LIN {X -0.262,Y -467.688,Z 682.023,A 0.000,B 0.000,C 90.000,E1 220.092} C_DIS
LIN {X -0.082,Y -463.648,Z 682.012,A 0.000,B 0.000,C 90.000,E1 218.177} C_DIS
LIN {X -0.203,Y -456.849,Z 681.993,A 0.000,B 0.000,C 90.000,E1 214.692} C_DIS
LIN {X -0.182,Y -453.797,Z 681.984,A 0.000,B 0.000,C 90.000,E1 213.086} C_DIS
LIN {X -0.004,Y -450.100,Z 681.973,A 0.000,B 0.000,C 90.000,E1 211.131} C_DIS
LIN {X -0.145,Y -446.430,Z 681.962,A 0.000,B 0.000,C 90.000,E1 209.205} C_DIS
LIN {X -0.102,Y -444.091,Z 681.955,A 0.000,B 0.000,C 90.000,E1 207.897} C_DIS
LIN {X 0.139,Y -441.158,Z 681.946,A 0.000,B 0.000,C 90.000,E1 206.232} C_DIS
LIN {X -0.011,Y -437.014,Z 681.933,A 0.000,B 0.000,C 90.000,E1 203.951} C_DIS
LIN {X -0.104,Y -434.577,Z 681.926,A 0.000,B 0.000,C 90.000,E1 202.642} C_DIS
LIN {X 0.163,Y -432.175,Z 681.918,A 0.000,B 0.000,C 90.000,E1 201.280} C_DIS
LIN {X -0.146,Y -428.524,Z 681.907,A 0.000,B 0.000,C 90.000,E1 199.322} C_DIS
LIN {X 0.126,Y -424.968,Z 681.896,A 0.000,B 0.000,C 90.000,E1 197.275} C_DIS
LIN {X -0.054,Y -422.696,Z 681.889,A 0.000,B 0.000,C 90.000,E1 195.953} C_DIS
LIN {X 0.018,Y -420.416,Z 681.881,A 0.000,B 0.000,C 90.000,E1 194.592} C_DIS
LIN {X -0.187,Y -416.227,Z 681.868,A 0.000,B 0.000,C 90.000,E1 192.243} C_DIS
LIN {X -0.218,Y -412.981,Z 681.857,A 0.000,B 0.000,C 90.000,E1 190.197} C_DIS
LIN {X 0.002,Y -409.736,Z 681.845,A 0.000,B 0.000,C 90.000,E1 188.106} C_DIS
LIN {X 0.030,Y -406.654,Z 681.834,A 0.000,B 0.000,C 90.000,E1 186.030} C_DIS
LIN {X -0.055,Y -403.359,Z 681.820,A 0.000,B 0.000,C 90.000,E1 183.612} C_DIS
LIN {X 0.066,Y -399.999,Z 681.805,A 0.000,B 0.000,C 90.000,E1 180.802} C_DIS
LIN {X -0.174,Y -398.274,Z 681.795,A 0.000,B 0.000,C 90.000,E1 179.083} C_DIS
LIN {X 0.076,Y -395.388,Z 681.775,A 0.000,B 0.000,C 90.000,E1 175.527} C_DIS
LIN {X -0.039,Y -393.501,Z 681.756,A 0.000,B 0.000,C 90.000,E1 172.008} C_DIS
LIN {X 0.074,Y -392.686,Z 681.742,A 0.000,B 0.000,C 90.000,E1 169.511} C_DIS
LIN {X -0.065,Y -392.443,Z 681.732,A 0.000,B 0.000,C 90.000,E1 167.757} C_DIS
LIN {X -0.118,Y -392.239,Z 681.726,A 0.000,B 0.000,C 90.000,E1 166.700} C_DIS
LIN {X -0.113,Y -391.949,Z 681.708,A 0.000,B 0.000,C 90.000,E1 163.504} C_DIS
LIN {X -0.086,Y -391.984,Z 681.693,A 0.000,B 0.000,C 90.000,E1 160.659} C_DIS
LIN {X -0.162,Y -392.122,Z 681.681,A 0.000,B 0.000,C 90.000,E1 158.539} C_DIS
LIN {X -0.009,Y -392.271,Z 681.671,A 0.000,B 0.000,C 90.000,E1 156.741} C_DIS
LIN {X -0.051,Y -392.492,Z 681.661,A 0.000,B 0.000,C 90.000,E1 154.973} C_DIS
LIN {X 0.167,Y -392.920,Z 681.645,A 0.000,B 0.000,C 90.000,E1 152.103} C_DIS
LIN {X 0.145,Y -393.343,Z 681.635,A 0.000,B 0.000,C 90.000,E1 150.333} C_DIS
LIN {X 0.053,Y -394.052,Z 681.622,A 0.000,B 0.000,C 90.000,E1 147.867} C_DIS
LIN {X -0.013,Y -394.937,Z 681.610,A 0.000,B 0.000,C 90.000,E1 145.754} C_DIS
LIN {X 0.119,Y -396.736,Z 681.592,A 0.000,B 0.000,C 90.000,E1 142.557} C_DIS
LIN {X 0.175,Y -398.215,Z 681.580,A 0.000,B 0.000,C 90.000,E1 140.436} C_DIS
LIN {X 0.215,Y -399.929,Z 681.569,A 0.000,B 0.000,C 90.000,E1 138.324} C_DIS
LIN {X -0.025,Y -401.747,Z 681.557,A 0.000,B 0.000,C 90.000,E1 136.257} C_DIS
LIN {X 0.018,Y -402.831,Z 681.551,A 0.000,B 0.000,C 90.000,E1 135.202} C_DIS
LIN {X -0.047,Y -403.717,Z 681.547,A 0.000,B 0.000,C 90.000,E1 134.514} C_DIS
LIN {X 0.182,Y -405.074,Z 681.543,A 0.000,B 0.000,C 90.000,E1 133.785} C_DIS
LIN {X -0.070,Y -406.688,Z 681.541,A 0.000,B 0.000,C 90.000,E1 133.299} C_DIS
LIN {X -0.007,Y -409.347,Z 681.538,A 0.000,B 0.000,C 90.000,E1 132.771} C_DIS
LIN {X -0.087,Y -410.504,Z 681.537,A 0.000,B 0.000,C 90.000,E1 132.609} C_DIS
LIN {X 0.023,Y -413.364,Z 681.535,A 0.000,B 0.000,C 90.000,E1 132.243} C_DIS
LIN {X 0.058,Y -416.509,Z 681.533,A 0.000,B 0.000,C 90.000,E1 131.919} C_DIS
LIN {X -0.066,Y -436.386,Z 681.523,A 0.000,B 0.000,C 90.000,E1 130.216} C_DIS
LIN {X 0.047,Y -450.507,Z 681.517,A 0.000,B 0.000,C 90.000,E1 129.072} C_DIS
LIN {X 0.003,Y -462.969,Z 681.512,A 0.000,B 0.000,C 90.000,E1 128.096} C_DIS
LIN {X 0.286,Y -470.488,Z 681.508,A 0.000,B 0.000,C 90.000,E1 127.443} C_DIS
LIN {X 0.145,Y -476.410,Z 681.505,A 0.000,B 0.000,C 90.000,E1 126.950} C_DIS
LIN {X -0.146,Y -485.103,Z 681.501,A 0.000,B 0.000,C 90.000,E1 126.217} C_DIS
LIN {X -0.022,Y -490.767,Z 681.498,A 0.000,B 0.000,C 90.000,E1 125.678} C_DIS
LIN {X -0.126,Y -500.553,Z 681.493,A 0.000,B 0.000,C 90.000,E1 124.739} C_DIS
LIN {X -0.228,Y -505.962,Z 681.490,A 0.000,B 0.000,C 90.000,E1 124.199} C_DIS
LIN {X -0.102,Y -509.796,Z 681.488,A 0.000,B 0.000,C 90.000,E1 123.785} C_DIS
LIN {X -0.050,Y -514.951,Z 681.485,A 0.000,B 0.000,C 90.000,E1 123.214} C_DIS
LIN {X 0.169,Y -518.880,Z 681.482,A 0.000,B 0.000,C 90.000,E1 122.752} C_DIS
LIN {X -0.203,Y -523.625,Z 681.479,A 0.000,B 0.000,C 90.000,E1 122.212} C_DIS
LIN {X -0.085,Y -527.803,Z 681.476,A 0.000,B 0.000,C 90.000,E1 121.671} C_DIS
LIN {X 0.139,Y -532.881,Z 681.472,A 0.000,B 0.000,C 90.000,E1 120.924} C_DIS
LIN {X -0.180,Y -536.619,Z 681.469,A 0.000,B 0.000,C 90.000,E1 120.384} C_DIS
LIN {X -0.145,Y -540.710,Z 681.465,A 0.000,B 0.000,C 90.000,E1 119.667} C_DIS
LIN {X 0.058,Y -543.789,Z 681.462,A 0.000,B 0.000,C 90.000,E1 119.077} C_DIS
LIN {X 0.037,Y -547.865,Z 681.457,A 0.000,B 0.000,C 90.000,E1 118.231} C_DIS
LIN {X 0.061,Y -551.684,Z 681.452,A 0.000,B 0.000,C 90.000,E1 117.385} C_DIS
LIN {X -0.020,Y -554.604,Z 681.448,A 0.000,B 0.000,C 90.000,E1 116.693} C_DIS
LIN {X -0.147,Y -558.920,Z 681.442,A 0.000,B 0.000,C 90.000,E1 115.591} C_DIS
LIN {X -0.264,Y -561.960,Z 681.438,A 0.000,B 0.000,C 90.000,E1 114.771} C_DIS
LIN {X 0.168,Y -564.717,Z 681.433,A 0.000,B 0.000,C 90.000,E1 113.898} C_DIS
LIN {X 0.114,Y -567.136,Z 681.428,A 0.000,B 0.000,C 90.000,E1 113.078} C_DIS
LIN {X -0.137,Y -569.261,Z 681.424,A 0.000,B 0.000,C 90.000,E1 112.280} C_DIS
LIN {X -0.154,Y -571.189,Z 681.419,A 0.000,B 0.000,C 90.000,E1 111.461} C_DIS
LIN {X 0.170,Y -572.898,Z 681.415,A 0.000,B 0.000,C 90.000,E1 110.610} C_DIS
LIN {X -0.026,Y -575.531,Z 681.407,A 0.000,B 0.000,C 90.000,E1 109.268} C_DIS
LIN {X -0.185,Y -578.080,Z 681.400,A 0.000,B 0.000,C 90.000,E1 107.928} C_DIS
LIN {X 0.067,Y -580.625,Z 681.392,A 0.000,B 0.000,C 90.000,E1 106.551} C_DIS
LIN {X 0.208,Y -583.058,Z 681.385,A 0.000,B 0.000,C 90.000,E1 105.190} C_DIS
LIN {X 0.073,Y -585.830,Z 681.376,A 0.000,B 0.000,C 90.000,E1 103.592} C_DIS
LIN {X -0.145,Y -588.553,Z 681.367,A 0.000,B 0.000,C 90.000,E1 102.007} C_DIS
LIN {X 0.267,Y -591.283,Z 681.358,A 0.000,B 0.000,C 90.000,E1 100.366} C_DIS
LIN {X 0.075,Y -593.090,Z 681.352,A 0.000,B 0.000,C 90.000,E1 99.321} C_DIS
LIN {X 0.099,Y -595.138,Z 681.344,A 0.000,B 0.000,C 90.000,E1 97.992} C_DIS
LIN {X -0.151,Y -597.385,Z 681.336,A 0.000,B 0.000,C 90.000,E1 96.429} C_DIS
LIN {X -0.119,Y -599.199,Z 681.328,A 0.000,B 0.000,C 90.000,E1 95.106} C_DIS
LIN {X 0.184,Y -601.110,Z 681.320,A 0.000,B 0.000,C 90.000,E1 93.498} C_DIS
LIN {X -0.253,Y -601.976,Z 681.315,A 0.000,B 0.000,C 90.000,E1 92.751} C_DIS
LIN {X -0.184,Y -603.181,Z 681.308,A 0.000,B 0.000,C 90.000,E1 91.432} C_DIS
LIN {X -0.108,Y -604.203,Z 681.301,A 0.000,B 0.000,C 90.000,E1 90.115} C_DIS
LIN {X -0.275,Y -604.751,Z 681.295,A 0.000,B 0.000,C 90.000,E1 89.083} C_DIS
LIN {X 0.184,Y -605.098,Z 681.289,A 0.000,B 0.000,C 90.000,E1 87.993} C_DIS
LIN {X 0.312,Y -605.458,Z 681.282,A 0.000,B 0.000,C 90.000,E1 86.674} C_DIS
LIN {X 0.138,Y -605.513,Z 681.273,A 0.000,B 0.000,C 90.000,E1 85.122} C_DIS
LIN {X 0.309,Y -605.356,Z 681.266,A 0.000,B 0.000,C 90.000,E1 83.799} C_DIS
LIN {X -0.058,Y -605.000,Z 681.258,A 0.000,B 0.000,C 90.000,E1 82.527} C_DIS
LIN {X 0.131,Y -604.672,Z 681.254,A 0.000,B 0.000,C 90.000,E1 81.724} C_DIS
LIN {X 0.115,Y -604.063,Z 681.248,A 0.000,B 0.000,C 90.000,E1 80.679} C_DIS
LIN {X 0.091,Y -603.100,Z 681.242,A 0.000,B 0.000,C 90.000,E1 79.634} C_DIS
LIN {X 0.167,Y -602.158,Z 681.237,A 0.000,B 0.000,C 90.000,E1 78.578} C_DIS
LIN {X 0.267,Y -600.426,Z 681.228,A 0.000,B 0.000,C 90.000,E1 76.992} C_DIS
LIN {X 0.027,Y -598.834,Z 681.221,A 0.000,B 0.000,C 90.000,E1 75.700} C_DIS
LIN {X -0.094,Y -597.145,Z 681.213,A 0.000,B 0.000,C 90.000,E1 74.393} C_DIS
LIN {X -0.248,Y -595.232,Z 681.206,A 0.000,B 0.000,C 90.000,E1 73.087} C_DIS
LIN {X 0.040,Y -593.634,Z 681.200,A 0.000,B 0.000,C 90.000,E1 72.000} C_DIS
LIN {X 0.306,Y -591.877,Z 681.194,A 0.000,B 0.000,C 90.000,E1 70.913} C_DIS
LIN {X -0.012,Y -590.024,Z 681.188,A 0.000,B 0.000,C 90.000,E1 69.880} C_DIS
LIN {X 0.065,Y -587.376,Z 681.181,A 0.000,B 0.000,C 90.000,E1 68.539} C_DIS
LIN {X -0.107,Y -584.949,Z 681.175,A 0.000,B 0.000,C 90.000,E1 67.486} C_DIS
LIN {X -0.080,Y -582.213,Z 681.169,A 0.000,B 0.000,C 90.000,E1 66.410} C_DIS
LIN {X -0.322,Y -579.130,Z 681.163,A 0.000,B 0.000,C 90.000,E1 65.357} C_DIS
LIN {X -0.222,Y -576.662,Z 681.158,A 0.000,B 0.000,C 90.000,E1 64.537} C_DIS
LIN {X 0.102,Y -573.960,Z 681.154,A 0.000,B 0.000,C 90.000,E1 63.691} C_DIS
LIN {X -0.022,Y -570.066,Z 681.148,A 0.000,B 0.000,C 90.000,E1 62.615} C_DIS
LIN {X 0.235,Y -566.949,Z 681.143,A 0.000,B 0.000,C 90.000,E1 61.769} C_DIS
LIN {X -0.125,Y -564.736,Z 681.140,A 0.000,B 0.000,C 90.000,E1 61.257} C_DIS
LIN {X 0.069,Y -561.100,Z 681.136,A 0.000,B 0.000,C 90.000,E1 60.411} C_DIS
LIN {X 0.014,Y -556.969,Z 681.131,A 0.000,B 0.000,C 90.000,E1 59.587} C_DIS
LIN {X 0.226,Y -553.041,Z 681.127,A 0.000,B 0.000,C 90.000,E1 58.869} C_DIS
LIN {X -0.072,Y -548.653,Z 681.123,A 0.000,B 0.000,C 90.000,E1 58.201} C_DIS
LIN {X -0.153,Y -545.872,Z 681.121,A 0.000,B 0.000,C 90.000,E1 57.788} C_DIS
LIN {X 0.078,Y -541.813,Z 681.118,A 0.000,B 0.000,C 90.000,E1 57.199} C_DIS
LIN {X 0.116,Y -537.275,Z 681.115,A 0.000,B 0.000,C 90.000,E1 56.628} C_DIS
LIN {X -0.097,Y -531.335,Z 681.111,A 0.000,B 0.000,C 90.000,E1 56.008} C_DIS
LIN {X 0.008,Y -527.377,Z 681.109,A 0.000,B 0.000,C 90.000,E1 55.595} C_DIS
LIN {X 0.042,Y -520.539,Z 681.106,A 0.000,B 0.000,C 90.000,E1 55.022} C_DIS
LIN {X 0.147,Y -517.509,Z 681.104,A 0.000,B 0.000,C 90.000,E1 54.769} C_DIS
LIN {X 0.004,Y -511.640,Z 681.102,A 0.000,B 0.000,C 90.000,E1 54.356} C_DIS
LIN {X 0.135,Y -503.729,Z 681.099,A 0.000,B 0.000,C 90.000,E1 53.829} C_DIS
LIN {X 0.237,Y -496.968,Z 681.097,A 0.000,B 0.000,C 90.000,E1 53.417} C_DIS
LIN {X 0.202,Y -490.450,Z 681.095,A 0.000,B 0.000,C 90.000,E1 53.050} C_DIS
LIN {X -0.149,Y -470.678,Z 681.089,A 0.000,B 0.000,C 90.000,E1 51.984} C_DIS
LIN {X -0.020,Y -452.548,Z 681.083,A 0.000,B 0.000,C 90.000,E1 50.928} C_DIS
LIN {X 0.018,Y -432.868,Z 681.076,A 0.000,B 0.000,C 90.000,E1 49.703} C_DIS
LIN {X -0.166,Y -427.914,Z 681.074,A 0.000,B 0.000,C 90.000,E1 49.380} C_DIS
LIN {X -0.193,Y -427.878,Z 681.074,A 0.000,B 0.000,C 90.000,E1 49.380} C_DIS
LIN {X -0.028,Y -418.736,Z 681.049,A 0.000,B 0.000,C 90.000,E1 44.879} C_DIS
LIN {X -0.117,Y -414.248,Z 681.038,A 0.000,B 0.000,C 90.000,E1 42.933} C_DIS
LIN {X -0.030,Y -414.313,Z 681.027,A 0.000,B 0.000,C 90.000,E1 40.782} C_DIS
LIN {X -0.053,Y -414.991,Z 681.008,A 0.000,B 0.000,C 90.000,E1 37.363} C_DIS
LIN {X -0.049,Y -415.932,Z 680.996,A 0.000,B 0.000,C 90.000,E1 35.311} C_DIS
LIN {X 0.192,Y -416.571,Z 680.989,A 0.000,B 0.000,C 90.000,E1 33.913} C_DIS
LIN {X 0.115,Y -417.667,Z 680.977,A 0.000,B 0.000,C 90.000,E1 31.878} C_DIS
LIN {X -0.111,Y -418.585,Z 680.968,A 0.000,B 0.000,C 90.000,E1 30.207} C_DIS
LIN {X -0.002,Y -419.762,Z 680.956,A 0.000,B 0.000,C 90.000,E1 28.153} C_DIS
LIN {X -0.121,Y -421.292,Z 680.943,A 0.000,B 0.000,C 90.000,E1 25.796} C_DIS
LIN {X -0.115,Y -424.378,Z 680.923,A 0.000,B 0.000,C 90.000,E1 22.078} C_DIS
LIN {X 0.032,Y -426.000,Z 680.913,A 0.000,B 0.000,C 90.000,E1 20.375} C_DIS
LIN {X -0.184,Y -427.522,Z 680.904,A 0.000,B 0.000,C 90.000,E1 18.725} C_DIS
LIN {X 0.101,Y -429.201,Z 680.893,A 0.000,B 0.000,C 90.000,E1 16.677} C_DIS
LIN {X 0.086,Y -430.760,Z 680.883,A 0.000,B 0.000,C 90.000,E1 15.009} C_DIS
LIN {X -0.104,Y -433.179,Z 680.871,A 0.000,B 0.000,C 90.000,E1 12.703} C_DIS
LIN {X 0.000,Y -435.741,Z 680.858,A 0.000,B 0.000,C 90.000,E1 10.366} C_DIS
LIN {X 0.177,Y -438.870,Z 680.843,A 0.000,B 0.000,C 90.000,E1 7.701} C_DIS
LIN {X 0.087,Y -441.395,Z 680.832,A 0.000,B 0.000,C 90.000,E1 5.739} C_DIS
LIN {X -0.022,Y -445.512,Z 680.816,A 0.000,B 0.000,C 90.000,E1 2.808} C_DIS
LIN {X -0.201,Y -449.595,Z 680.801,A 0.000,B 0.000,C 90.000,E1 0.229} C_DIS
LIN {X 0.146,Y -454.849,Z 680.785,A 0.000,B 0.000,C 90.000,E1 357.192} C_DIS
LIN {X -0.214,Y -456.662,Z 680.779,A 0.000,B 0.000,C 90.000,E1 356.274} C_DIS
LIN {X 0.077,Y -460.316,Z 680.769,A 0.000,B 0.000,C 90.000,E1 354.318} C_DIS
LIN {X -0.205,Y -463.319,Z 680.760,A 0.000,B 0.000,C 90.000,E1 352.761} C_DIS
LIN {X -0.104,Y -466.928,Z 680.749,A 0.000,B 0.000,C 90.000,E1 350.849} C_DIS
LIN {X -0.121,Y -469.814,Z 680.740,A 0.000,B 0.000,C 90.000,E1 349.275} C_DIS
LIN {X 0.205,Y -473.113,Z 680.730,A 0.000,B 0.000,C 90.000,E1 347.353} C_DIS
LIN {X -0.069,Y -475.935,Z 680.721,A 0.000,B 0.000,C 90.000,E1 345.825} C_DIS
LIN {X 0.099,Y -480.046,Z 680.709,A 0.000,B 0.000,C 90.000,E1 343.630} C_DIS
LIN {X 0.199,Y -483.621,Z 680.699,A 0.000,B 0.000,C 90.000,E1 341.764} C_DIS
LIN {X 0.086,Y -487.393,Z 680.689,A 0.000,B 0.000,C 90.000,E1 339.934} C_DIS
LIN {X 0.030,Y -490.524,Z 680.680,A 0.000,B 0.000,C 90.000,E1 338.411} C_DIS
LIN {X -0.211,Y -494.142,Z 680.670,A 0.000,B 0.000,C 90.000,E1 336.613} C_DIS
LIN {X 0.090,Y -498.384,Z 680.658,A 0.000,B 0.000,C 90.000,E1 334.460} C_DIS
LIN {X -0.248,Y -499.943,Z 680.655,A 0.000,B 0.000,C 90.000,E1 333.896} C_DIS
LIN {X 0.032,Y -500.860,Z 680.653,A 0.000,B 0.000,C 90.000,E1 333.563} C_DIS
LIN {X 0.093,Y -502.010,Z 680.652,A 0.000,B 0.000,C 90.000,E1 333.256} C_DIS
LIN {X 0.155,Y -503.590,Z 680.650,A 0.000,B 0.000,C 90.000,E1 332.948} C_DIS
LIN {X 0.081,Y -508.354,Z 680.647,A 0.000,B 0.000,C 90.000,E1 332.359} C_DIS
LIN {X -0.103,Y -509.791,Z 680.646,A 0.000,B 0.000,C 90.000,E1 332.231} C_DIS
LIN {X -0.067,Y -515.345,Z 680.643,A 0.000,B 0.000,C 90.000,E1 331.769} C_DIS
LIN {X -0.177,Y -520.162,Z 680.641,A 0.000,B 0.000,C 90.000,E1 331.435} C_DIS
LIN {X 0.088,Y -531.053,Z 680.637,A 0.000,B 0.000,C 90.000,E1 330.667} C_DIS
LIN {X 0.134,Y -538.647,Z 680.634,A 0.000,B 0.000,C 90.000,E1 330.127} C_DIS
LIN {X 0.142,Y -543.018,Z 680.632,A 0.000,B 0.000,C 90.000,E1 329.793} C_DIS
LIN {X -0.204,Y -551.551,Z 680.628,A 0.000,B 0.000,C 90.000,E1 329.125} C_DIS
LIN {X 0.055,Y -557.054,Z 680.626,A 0.000,B 0.000,C 90.000,E1 328.614} C_DIS
LIN {X -0.119,Y -563.731,Z 680.622,A 0.000,B 0.000,C 90.000,E1 327.995} C_DIS
LIN {X -0.257,Y -571.536,Z 680.618,A 0.000,B 0.000,C 90.000,E1 327.248} C_DIS
LIN {X 0.092,Y -581.679,Z 680.612,A 0.000,B 0.000,C 90.000,E1 326.167} C_DIS
LIN {X 0.240,Y -591.700,Z 680.606,A 0.000,B 0.000,C 90.000,E1 325.102} C_DIS
LIN {X -0.129,Y -597.822,Z 680.603,A 0.000,B 0.000,C 90.000,E1 324.482} C_DIS
LIN {X -0.092,Y -604.517,Z 680.598,A 0.000,B 0.000,C 90.000,E1 323.703} C_DIS
LIN {X -0.146,Y -610.993,Z 680.594,A 0.000,B 0.000,C 90.000,E1 322.924} C_DIS
LIN {X -0.279,Y -614.012,Z 680.592,A 0.000,B 0.000,C 90.000,E1 322.557} C_DIS
LIN {X -0.074,Y -617.805,Z 680.589,A 0.000,B 0.000,C 90.000,E1 322.029} C_DIS
LIN {X 0.078,Y -624.202,Z 680.584,A 0.000,B 0.000,C 90.000,E1 321.126} C_DIS
LIN {X 0.124,Y -629.303,Z 680.580,A 0.000,B 0.000,C 90.000,E1 320.356} C_DIS
LIN {X -0.136,Y -634.087,Z 680.576,A 0.000,B 0.000,C 90.000,E1 319.622} C_DIS
LIN {X -0.002,Y -639.506,Z 680.571,A 0.000,B 0.000,C 90.000,E1 318.728} C_DIS
LIN {X 0.071,Y -646.020,Z 680.565,A 0.000,B 0.000,C 90.000,E1 317.595} C_DIS
LIN {X -0.146,Y -651.483,Z 680.559,A 0.000,B 0.000,C 90.000,E1 316.620} C_DIS
LIN {X -0.327,Y -656.634,Z 680.553,A 0.000,B 0.000,C 90.000,E1 315.648} C_DIS
LIN {X 0.012,Y -661.902,Z 680.547,A 0.000,B 0.000,C 90.000,E1 314.514} C_DIS
LIN {X -0.050,Y -669.447,Z 680.538,A 0.000,B 0.000,C 90.000,E1 312.813} C_DIS
LIN {X 0.040,Y -674.577,Z 680.531,A 0.000,B 0.000,C 90.000,E1 311.595} C_DIS
LIN {X 0.167,Y -677.481,Z 680.527,A 0.000,B 0.000,C 90.000,E1 310.862} C_DIS
LIN {X -0.158,Y -681.057,Z 680.522,A 0.000,B 0.000,C 90.000,E1 309.930} C_DIS
LIN {X 0.038,Y -683.464,Z 680.518,A 0.000,B 0.000,C 90.000,E1 309.197} C_DIS
LIN {X 0.260,Y -685.672,Z 680.514,A 0.000,B 0.000,C 90.000,E1 308.463} C_DIS
LIN {X 0.129,Y -688.345,Z 680.509,A 0.000,B 0.000,C 90.000,E1 307.523} C_DIS
LIN {X 0.029,Y -690.746,Z 680.503,A 0.000,B 0.000,C 90.000,E1 306.583} C_DIS
LIN {X -0.092,Y -692.377,Z 680.499,A 0.000,B 0.000,C 90.000,E1 305.884} C_DIS
LIN {X -0.151,Y -694.351,Z 680.494,A 0.000,B 0.000,C 90.000,E1 304.945} C_DIS
LIN {X -0.014,Y -696.083,Z 680.489,A 0.000,B 0.000,C 90.000,E1 303.992} C_DIS
LIN {X -0.188,Y -697.946,Z 680.482,A 0.000,B 0.000,C 90.000,E1 302.832} C_DIS
LIN {X -0.080,Y -699.754,Z 680.475,A 0.000,B 0.000,C 90.000,E1 301.416} C_DIS
LIN {X -0.134,Y -700.537,Z 680.471,A 0.000,B 0.000,C 90.000,E1 300.718} C_DIS
LIN {X -0.009,Y -701.544,Z 680.464,A 0.000,B 0.000,C 90.000,E1 299.539} C_DIS
LIN {X -0.140,Y -702.185,Z 680.459,A 0.000,B 0.000,C 90.000,E1 298.615} C_DIS
LIN {X -0.376,Y -703.277,Z 680.450,A 0.000,B 0.000,C 90.000,E1 297.001} C_DIS
LIN {X 0.101,Y -704.108,Z 680.443,A 0.000,B 0.000,C 90.000,E1 295.796} C_DIS
LIN {X -0.248,Y -704.176,Z 680.442,A 0.000,B 0.000,C 90.000,E1 295.591} C_DIS
LIN {X 0.321,Y -703.883,Z 680.440,A 0.000,B 0.000,C 90.000,E1 295.079} C_DIS
LIN {X -0.330,Y -703.415,Z 680.438,A 0.000,B 0.000,C 90.000,E1 294.899} C_DIS
LIN {X 0.235,Y -701.725,Z 680.436,A 0.000,B 0.000,C 90.000,E1 294.387} C_DIS
LIN {X 0.084,Y -701.161,Z 680.435,A 0.000,B 0.000,C 90.000,E1 294.283} C_DIS
LIN {X 0.224,Y -700.294,Z 680.434,A 0.000,B 0.000,C 90.000,E1 294.155} C_DIS
LIN {X 0.034,Y -696.602,Z 680.432,A 0.000,B 0.000,C 90.000,E1 293.823} C_DIS
LIN {X 0.227,Y -693.623,Z 680.431,A 0.000,B 0.000,C 90.000,E1 293.590} C_DIS
LIN {X -0.111,Y -691.217,Z 680.431,A 0.000,B 0.000,C 90.000,E1 293.515} C_DIS
LIN {X -0.052,Y -689.267,Z 680.430,A 0.000,B 0.000,C 90.000,E1 293.439} C_DIS
LIN {X -0.242,Y -684.728,Z 680.430,A 0.000,B 0.000,C 90.000,E1 293.334} C_DIS
LIN {X 0.184,Y -680.609,Z 680.429,A 0.000,B 0.000,C 90.000,E1 293.206} C_DIS
LIN {X -0.310,Y -678.138,Z 680.429,A 0.000,B 0.000,C 90.000,E1 293.206} C_DIS
LIN {X 0.089,Y -665.489,Z 680.428,A 0.000,B 0.000,C 90.000,E1 293.025} C_DIS
LIN {X 0.164,Y -651.606,Z 680.427,A 0.000,B 0.000,C 90.000,E1 292.823} C_DIS
LIN {X 0.053,Y -638.429,Z 680.426,A 0.000,B 0.000,C 90.000,E1 292.589} C_DIS
LIN {X -0.125,Y -628.350,Z 680.424,A 0.000,B 0.000,C 90.000,E1 292.386} C_DIS
LIN {X -0.270,Y -618.553,Z 680.423,A 0.000,B 0.000,C 90.000,E1 292.153} C_DIS
LIN {X -0.017,Y -597.959,Z 680.420,A 0.000,B 0.000,C 90.000,E1 291.535} C_DIS
LIN {X 0.176,Y -577.183,Z 680.416,A 0.000,B 0.000,C 90.000,E1 290.865} C_DIS
LIN {X -0.157,Y -562.746,Z 680.414,A 0.000,B 0.000,C 90.000,E1 290.482} C_DIS
LIN {X 0.066,Y -557.078,Z 680.412,A 0.000,B 0.000,C 90.000,E1 290.194} C_DIS
LIN {X 0.304,Y -555.465,Z 680.411,A 0.000,B 0.000,C 90.000,E1 289.993} C_DIS
LIN {X 0.263,Y -555.446,Z 680.411,A 0.000,B 0.000,C 90.000,E1 289.993} C_DIS
LIN {X -0.024,Y -554.607,Z 680.409,A 0.000,B 0.000,C 90.000,E1 289.704} C_DIS
LIN {X -0.279,Y -554.200,Z 680.406,A 0.000,B 0.000,C 90.000,E1 289.033} C_DIS
LIN {X 0.140,Y -553.933,Z 680.399,A 0.000,B 0.000,C 90.000,E1 287.873} C_DIS
LIN {X -0.193,Y -553.346,Z 680.389,A 0.000,B 0.000,C 90.000,E1 285.953} C_DIS
LIN {X 0.113,Y -552.702,Z 680.379,A 0.000,B 0.000,C 90.000,E1 284.245} C_DIS
LIN {X 0.181,Y -552.179,Z 680.373,A 0.000,B 0.000,C 90.000,E1 283.119} C_DIS
LIN {X 0.231,Y -551.453,Z 680.365,A 0.000,B 0.000,C 90.000,E1 281.715} C_DIS
LIN {X 0.154,Y -550.922,Z 680.359,A 0.000,B 0.000,C 90.000,E1 280.602} C_DIS
LIN {X 0.299,Y -550.054,Z 680.348,A 0.000,B 0.000,C 90.000,E1 278.624} C_DIS
LIN {X -0.181,Y -549.531,Z 680.336,A 0.000,B 0.000,C 90.000,E1 276.429} C_DIS
LIN {X 0.222,Y -549.287,Z 680.326,A 0.000,B 0.000,C 90.000,E1 274.702} C_DIS
LIN {X -0.055,Y -549.213,Z 680.318,A 0.000,B 0.000,C 90.000,E1 273.326} C_DIS
LIN {X 0.227,Y -548.968,Z 680.311,A 0.000,B 0.000,C 90.000,E1 271.892} C_DIS
LIN {X -0.050,Y -548.400,Z 680.303,A 0.000,B 0.000,C 90.000,E1 270.516} C_DIS
LIN {X 0.197,Y -547.576,Z 680.295,A 0.000,B 0.000,C 90.000,E1 269.083} C_DIS
LIN {X -0.023,Y -546.444,Z 680.284,A 0.000,B 0.000,C 90.000,E1 267.135} C_DIS
LIN {X 0.157,Y -545.695,Z 680.278,A 0.000,B 0.000,C 90.000,E1 265.988} C_DIS
LIN {X -0.074,Y -544.422,Z 680.268,A 0.000,B 0.000,C 90.000,E1 264.318} C_DIS
LIN {X 0.121,Y -543.459,Z 680.262,A 0.000,B 0.000,C 90.000,E1 263.166} C_DIS
LIN {X -0.168,Y -541.934,Z 680.254,A 0.000,B 0.000,C 90.000,E1 261.781} C_DIS
LIN {X -0.108,Y -539.447,Z 680.240,A 0.000,B 0.000,C 90.000,E1 259.218} C_DIS
LIN {X 0.247,Y -538.204,Z 680.232,A 0.000,B 0.000,C 90.000,E1 257.757} C_DIS
LIN {X 0.104,Y -536.815,Z 680.223,A 0.000,B 0.000,C 90.000,E1 256.061} C_DIS
LIN {X 0.132,Y -535.568,Z 680.215,A 0.000,B 0.000,C 90.000,E1 254.629} C_DIS
LIN {X -0.129,Y -533.506,Z 680.204,A 0.000,B 0.000,C 90.000,E1 252.653} C_DIS
LIN {X -0.260,Y -531.228,Z 680.191,A 0.000,B 0.000,C 90.000,E1 250.369} C_DIS
LIN {X -0.180,Y -529.817,Z 680.184,A 0.000,B 0.000,C 90.000,E1 249.209} C_DIS
LIN {X 0.071,Y -528.258,Z 680.178,A 0.000,B 0.000,C 90.000,E1 248.028} C_DIS
LIN {X -0.040,Y -525.730,Z 680.168,A 0.000,B 0.000,C 90.000,E1 246.305} C_DIS
LIN {X 0.204,Y -522.795,Z 680.159,A 0.000,B 0.000,C 90.000,E1 244.537} C_DIS
LIN {X -0.052,Y -521.240,Z 680.154,A 0.000,B 0.000,C 90.000,E1 243.691} C_DIS
LIN {X -0.010,Y -517.226,Z 680.143,A 0.000,B 0.000,C 90.000,E1 241.641} C_DIS
LIN {X 0.041,Y -514.834,Z 680.136,A 0.000,B 0.000,C 90.000,E1 240.461} C_DIS
LIN {X -0.054,Y -510.405,Z 680.125,A 0.000,B 0.000,C 90.000,E1 238.408} C_DIS
LIN {X 0.048,Y -507.108,Z 680.116,A 0.000,B 0.000,C 90.000,E1 236.914} C_DIS
LIN {X -0.049,Y -503.662,Z 680.108,A 0.000,B 0.000,C 90.000,E1 235.435} C_DIS
LIN {X -0.082,Y -500.812,Z 680.101,A 0.000,B 0.000,C 90.000,E1 234.242} C_DIS
LIN {X 0.108,Y -497.101,Z 680.093,A 0.000,B 0.000,C 90.000,E1 232.718} C_DIS
LIN {X -0.269,Y -493.416,Z 680.085,A 0.000,B 0.000,C 90.000,E1 231.251} C_DIS
LIN {X 0.136,Y -489.025,Z 680.074,A 0.000,B 0.000,C 90.000,E1 229.380} C_DIS
LIN {X 0.069,Y -484.708,Z 680.064,A 0.000,B 0.000,C 90.000,E1 227.553} C_DIS
LIN {X -0.124,Y -480.350,Z 680.054,A 0.000,B 0.000,C 90.000,E1 225.729} C_DIS
LIN {X 0.028,Y -477.482,Z 680.047,A 0.000,B 0.000,C 90.000,E1 224.474} C_DIS
LIN {X 0.110,Y -472.435,Z 680.035,A 0.000,B 0.000,C 90.000,E1 222.285} C_DIS
LIN {X 0.101,Y -467.688,Z 680.023,A 0.000,B 0.000,C 90.000,E1 220.092} C_DIS
LIN {X -0.087,Y -463.652,Z 680.012,A 0.000,B 0.000,C 90.000,E1 218.222} C_DIS
LIN {X -0.070,Y -458.542,Z 679.998,A 0.000,B 0.000,C 90.000,E1 215.678} C_DIS
LIN {X -0.117,Y -456.238,Z 679.991,A 0.000,B 0.000,C 90.000,E1 214.405} C_DIS
LIN {X 0.171,Y -453.798,Z 679.984,A 0.000,B 0.000,C 90.000,E1 213.086} C_DIS
LIN {X 0.258,Y -450.731,Z 679.975,A 0.000,B 0.000,C 90.000,E1 211.465} C_DIS
LIN {X 0.130,Y -447.065,Z 679.964,A 0.000,B 0.000,C 90.000,E1 209.539} C_DIS
LIN {X 0.244,Y -444.112,Z 679.955,A 0.000,B 0.000,C 90.000,E1 207.897} C_DIS
LIN {X 0.086,Y -441.179,Z 679.946,A 0.000,B 0.000,C 90.000,E1 206.283} C_DIS
LIN {X -0.086,Y -437.602,Z 679.935,A 0.000,B 0.000,C 90.000,E1 204.335} C_DIS
LIN {X -0.167,Y -435.226,Z 679.928,A 0.000,B 0.000,C 90.000,E1 203.025} C_DIS
LIN {X -0.058,Y -432.214,Z 679.919,A 0.000,B 0.000,C 90.000,E1 201.354} C_DIS
LIN {X 0.189,Y -428.567,Z 679.908,A 0.000,B 0.000,C 90.000,E1 199.322} C_DIS
LIN {X 0.054,Y -425.012,Z 679.896,A 0.000,B 0.000,C 90.000,E1 197.330} C_DIS
LIN {X -0.063,Y -422.176,Z 679.887,A 0.000,B 0.000,C 90.000,E1 195.662} C_DIS
LIN {X 0.005,Y -419.852,Z 679.880,A 0.000,B 0.000,C 90.000,E1 194.300} C_DIS
LIN {X 0.144,Y -416.303,Z 679.868,A 0.000,B 0.000,C 90.000,E1 192.243} C_DIS
LIN {X 0.112,Y -413.066,Z 679.857,A 0.000,B 0.000,C 90.000,E1 190.197} C_DIS
LIN {X -0.105,Y -410.380,Z 679.847,A 0.000,B 0.000,C 90.000,E1 188.511} C_DIS
LIN {X -0.015,Y -407.258,Z 679.836,A 0.000,B 0.000,C 90.000,E1 186.429} C_DIS
LIN {X -0.128,Y -403.458,Z 679.820,A 0.000,B 0.000,C 90.000,E1 183.669} C_DIS
LIN {X -0.005,Y -400.118,Z 679.805,A 0.000,B 0.000,C 90.000,E1 180.859} C_DIS
LIN {X 0.104,Y -398.064,Z 679.793,A 0.000,B 0.000,C 90.000,E1 178.740} C_DIS
LIN {X -0.056,Y -395.278,Z 679.774,A 0.000,B 0.000,C 90.000,E1 175.241} C_DIS
LIN {X -0.053,Y -393.783,Z 679.758,A 0.000,B 0.000,C 90.000,E1 172.413} C_DIS
LIN {X 0.000,Y -392.937,Z 679.744,A 0.000,B 0.000,C 90.000,E1 169.926} C_DIS
LIN {X -0.150,Y -392.517,Z 679.730,A 0.000,B 0.000,C 90.000,E1 167.465} C_DIS
LIN {X -0.175,Y -392.133,Z 679.715,A 0.000,B 0.000,C 90.000,E1 164.629} C_DIS
LIN {X -0.039,Y -392.092,Z 679.705,A 0.000,B 0.000,C 90.000,E1 162.834} C_DIS
LIN {X -0.181,Y -392.191,Z 679.691,A 0.000,B 0.000,C 90.000,E1 160.369} C_DIS
LIN {X 0.073,Y -392.437,Z 679.677,A 0.000,B 0.000,C 90.000,E1 157.847} C_DIS
LIN {X 0.118,Y -392.668,Z 679.663,A 0.000,B 0.000,C 90.000,E1 155.357} C_DIS
LIN {X 0.138,Y -393.073,Z 679.649,A 0.000,B 0.000,C 90.000,E1 152.871} C_DIS
LIN {X -0.209,Y -393.526,Z 679.638,A 0.000,B 0.000,C 90.000,E1 150.795} C_DIS
LIN {X -0.158,Y -394.032,Z 679.626,A 0.000,B 0.000,C 90.000,E1 148.663} C_DIS
LIN {X 0.058,Y -395.151,Z 679.610,A 0.000,B 0.000,C 90.000,E1 145.801} C_DIS
LIN {X -0.029,Y -396.898,Z 679.592,A 0.000,B 0.000,C 90.000,E1 142.637} C_DIS
LIN {X 0.133,Y -398.575,Z 679.579,A 0.000,B 0.000,C 90.000,E1 140.150} C_DIS
LIN {X -0.012,Y -400.583,Z 679.565,A 0.000,B 0.000,C 90.000,E1 137.715} C_DIS
LIN {X -0.241,Y -402.324,Z 679.553,A 0.000,B 0.000,C 90.000,E1 135.648} C_DIS
LIN {X -0.197,Y -403.488,Z 679.548,A 0.000,B 0.000,C 90.000,E1 134.595} C_DIS
LIN {X -0.040,Y -405.005,Z 679.543,A 0.000,B 0.000,C 90.000,E1 133.704} C_DIS
LIN {X -0.079,Y -407.129,Z 679.539,A 0.000,B 0.000,C 90.000,E1 133.014} C_DIS
LIN {X -0.243,Y -408.944,Z 679.537,A 0.000,B 0.000,C 90.000,E1 132.690} C_DIS
LIN {X -0.022,Y -409.994,Z 679.536,A 0.000,B 0.000,C 90.000,E1 132.486} C_DIS
LIN {X -0.056,Y -412.778,Z 679.534,A 0.000,B 0.000,C 90.000,E1 132.123} C_DIS
LIN {X -0.052,Y -418.107,Z 679.531,A 0.000,B 0.000,C 90.000,E1 131.595} C_DIS
LIN {X 0.007,Y -432.160,Z 679.524,A 0.000,B 0.000,C 90.000,E1 130.378} C_DIS
LIN {X -0.001,Y -447.958,Z 679.517,A 0.000,B 0.000,C 90.000,E1 129.116} C_DIS
LIN {X 0.006,Y -463.555,Z 679.511,A 0.000,B 0.000,C 90.000,E1 127.890} C_DIS
LIN {X -0.081,Y -471.066,Z 679.507,A 0.000,B 0.000,C 90.000,E1 127.282} C_DIS
LIN {X 0.015,Y -480.054,Z 679.503,A 0.000,B 0.000,C 90.000,E1 126.503} C_DIS
LIN {X -0.196,Y -485.849,Z 679.500,A 0.000,B 0.000,C 90.000,E1 126.011} C_DIS
LIN {X 0.106,Y -492.938,Z 679.496,A 0.000,B 0.000,C 90.000,E1 125.311} C_DIS
LIN {X 0.293,Y -499.996,Z 679.493,A 0.000,B 0.000,C 90.000,E1 124.612} C_DIS
LIN {X -0.188,Y -505.450,Z 679.490,A 0.000,B 0.000,C 90.000,E1 124.119} C_DIS
LIN {X 0.237,Y -512.118,Z 679.486,A 0.000,B 0.000,C 90.000,E1 123.372} C_DIS
LIN {X 0.103,Y -518.627,Z 679.482,A 0.000,B 0.000,C 90.000,E1 122.673} C_DIS
LIN {X 0.119,Y -525.774,Z 679.477,A 0.000,B 0.000,C 90.000,E1 121.799} C_DIS
LIN {X -0.114,Y -527.982,Z 679.475,A 0.000,B 0.000,C 90.000,E1 121.544} C_DIS
LIN {X -0.184,Y -532.796,Z 679.471,A 0.000,B 0.000,C 90.000,E1 120.875} C_DIS
LIN {X -0.254,Y -536.437,Z 679.468,A 0.000,B 0.000,C 90.000,E1 120.335} C_DIS
LIN {X -0.086,Y -539.858,Z 679.465,A 0.000,B 0.000,C 90.000,E1 119.745} C_DIS
LIN {X -0.017,Y -543.760,Z 679.461,A 0.000,B 0.000,C 90.000,E1 119.027} C_DIS
LIN {X 0.119,Y -547.861,Z 679.457,A 0.000,B 0.000,C 90.000,E1 118.180} C_DIS
LIN {X 0.146,Y -551.715,Z 679.452,A 0.000,B 0.000,C 90.000,E1 117.334} C_DIS
LIN {X -0.175,Y -554.669,Z 679.448,A 0.000,B 0.000,C 90.000,E1 116.668} C_DIS
LIN {X 0.162,Y -557.974,Z 679.443,A 0.000,B 0.000,C 90.000,E1 115.796} C_DIS
LIN {X 0.042,Y -561.114,Z 679.439,A 0.000,B 0.000,C 90.000,E1 114.975} C_DIS
LIN {X -0.045,Y -563.981,Z 679.434,A 0.000,B 0.000,C 90.000,E1 114.155} C_DIS
LIN {X -0.105,Y -566.544,Z 679.430,A 0.000,B 0.000,C 90.000,E1 113.334} C_DIS
LIN {X -0.144,Y -568.793,Z 679.425,A 0.000,B 0.000,C 90.000,E1 112.514} C_DIS
LIN {X 0.151,Y -570.861,Z 679.420,A 0.000,B 0.000,C 90.000,E1 111.663} C_DIS
LIN {X -0.057,Y -572.645,Z 679.416,A 0.000,B 0.000,C 90.000,E1 110.865} C_DIS
LIN {X -0.060,Y -575.356,Z 679.408,A 0.000,B 0.000,C 90.000,E1 109.504} C_DIS
LIN {X -0.032,Y -578.432,Z 679.399,A 0.000,B 0.000,C 90.000,E1 107.873} C_DIS
LIN {X 0.231,Y -581.008,Z 679.392,A 0.000,B 0.000,C 90.000,E1 106.496} C_DIS
LIN {X -0.179,Y -583.477,Z 679.384,A 0.000,B 0.000,C 90.000,E1 105.190} C_DIS
LIN {X 0.018,Y -585.817,Z 679.377,A 0.000,B 0.000,C 90.000,E1 103.828} C_DIS
LIN {X -0.198,Y -588.593,Z 679.368,A 0.000,B 0.000,C 90.000,E1 102.243} C_DIS
LIN {X 0.219,Y -591.335,Z 679.359,A 0.000,B 0.000,C 90.000,E1 100.602} C_DIS
LIN {X 0.030,Y -593.198,Z 679.353,A 0.000,B 0.000,C 90.000,E1 99.557} C_DIS
LIN {X 0.144,Y -595.318,Z 679.346,A 0.000,B 0.000,C 90.000,E1 98.219} C_DIS
LIN {X -0.076,Y -596.850,Z 679.340,A 0.000,B 0.000,C 90.000,E1 97.182} C_DIS
LIN {X 0.012,Y -598.742,Z 679.333,A 0.000,B 0.000,C 90.000,E1 95.853} C_DIS
LIN {X -0.217,Y -600.191,Z 679.327,A 0.000,B 0.000,C 90.000,E1 94.821} C_DIS
LIN {X 0.113,Y -602.080,Z 679.318,A 0.000,B 0.000,C 90.000,E1 93.212} C_DIS
LIN {X 0.194,Y -603.388,Z 679.311,A 0.000,B 0.000,C 90.000,E1 91.892} C_DIS
LIN {X 0.290,Y -604.458,Z 679.303,A 0.000,B 0.000,C 90.000,E1 90.573} C_DIS
LIN {X 0.128,Y -605.154,Z 679.298,A 0.000,B 0.000,C 90.000,E1 89.542} C_DIS
LIN {X -0.029,Y -605.626,Z 679.292,A 0.000,B 0.000,C 90.000,E1 88.511} C_DIS
LIN {X -0.244,Y -606.038,Z 679.283,A 0.000,B 0.000,C 90.000,E1 86.963} C_DIS
LIN {X 0.274,Y -606.128,Z 679.277,A 0.000,B 0.000,C 90.000,E1 85.869} C_DIS
LIN {X -0.202,Y -606.094,Z 679.270,A 0.000,B 0.000,C 90.000,E1 84.609} C_DIS
LIN {X 0.035,Y -605.811,Z 679.263,A 0.000,B 0.000,C 90.000,E1 83.280} C_DIS
LIN {X 0.275,Y -605.376,Z 679.255,A 0.000,B 0.000,C 90.000,E1 81.951} C_DIS
LIN {X -0.098,Y -604.590,Z 679.248,A 0.000,B 0.000,C 90.000,E1 80.679} C_DIS
LIN {X 0.268,Y -603.885,Z 679.244,A 0.000,B 0.000,C 90.000,E1 79.859} C_DIS
LIN {X 0.284,Y -602.377,Z 679.235,A 0.000,B 0.000,C 90.000,E1 78.285} C_DIS
LIN {X 0.079,Y -600.849,Z 679.228,A 0.000,B 0.000,C 90.000,E1 76.992} C_DIS
LIN {X 0.144,Y -598.885,Z 679.219,A 0.000,B 0.000,C 90.000,E1 75.408} C_DIS
LIN {X -0.267,Y -597.495,Z 679.213,A 0.000,B 0.000,C 90.000,E1 74.393} C_DIS
LIN {X 0.032,Y -595.158,Z 679.204,A 0.000,B 0.000,C 90.000,E1 72.779} C_DIS
LIN {X 0.016,Y -593.019,Z 679.197,A 0.000,B 0.000,C 90.000,E1 71.456} C_DIS
LIN {X 0.154,Y -590.673,Z 679.190,A 0.000,B 0.000,C 90.000,E1 70.115} C_DIS
LIN {X -0.059,Y -589.136,Z 679.185,A 0.000,B 0.000,C 90.000,E1 69.337} C_DIS
LIN {X -0.207,Y -586.870,Z 679.179,A 0.000,B 0.000,C 90.000,E1 68.284} C_DIS
LIN {X -0.255,Y -584.998,Z 679.175,A 0.000,B 0.000,C 90.000,E1 67.486} C_DIS
LIN {X 0.308,Y -582.202,Z 679.169,A 0.000,B 0.000,C 90.000,E1 66.357} C_DIS
LIN {X 0.058,Y -579.042,Z 679.163,A 0.000,B 0.000,C 90.000,E1 65.305} C_DIS
LIN {X 0.151,Y -576.512,Z 679.158,A 0.000,B 0.000,C 90.000,E1 64.485} C_DIS
LIN {X -0.046,Y -573.750,Z 679.154,A 0.000,B 0.000,C 90.000,E1 63.691} C_DIS
LIN {X -0.171,Y -569.778,Z 679.148,A 0.000,B 0.000,C 90.000,E1 62.615} C_DIS
LIN {X 0.258,Y -567.721,Z 679.145,A 0.000,B 0.000,C 90.000,E1 62.025} C_DIS
LIN {X -0.100,Y -563.720,Z 679.139,A 0.000,B 0.000,C 90.000,E1 61.101} C_DIS
LIN {X -0.092,Y -560.584,Z 679.136,A 0.000,B 0.000,C 90.000,E1 60.411} C_DIS
LIN {X -0.048,Y -557.091,Z 679.132,A 0.000,B 0.000,C 90.000,E1 59.715} C_DIS
LIN {X 0.168,Y -553.109,Z 679.128,A 0.000,B 0.000,C 90.000,E1 58.997} C_DIS
LIN {X -0.009,Y -549.623,Z 679.125,A 0.000,B 0.000,C 90.000,E1 58.456} C_DIS
LIN {X -0.246,Y -544.906,Z 679.121,A 0.000,B 0.000,C 90.000,E1 57.788} C_DIS
LIN {X -0.144,Y -541.024,Z 679.118,A 0.000,B 0.000,C 90.000,E1 57.248} C_DIS
LIN {X 0.342,Y -536.361,Z 679.115,A 0.000,B 0.000,C 90.000,E1 56.628} C_DIS
LIN {X 0.190,Y -531.050,Z 679.112,A 0.000,B 0.000,C 90.000,E1 56.087} C_DIS
LIN {X -0.166,Y -526.969,Z 679.109,A 0.000,B 0.000,C 90.000,E1 55.722} C_DIS
LIN {X 0.178,Y -520.889,Z 679.107,A 0.000,B 0.000,C 90.000,E1 55.182} C_DIS
LIN {X -0.052,Y -514.616,Z 679.104,A 0.000,B 0.000,C 90.000,E1 54.736} C_DIS
LIN {X -0.032,Y -509.884,Z 679.102,A 0.000,B 0.000,C 90.000,E1 54.402} C_DIS
LIN {X 0.047,Y -503.456,Z 679.100,A 0.000,B 0.000,C 90.000,E1 53.989} C_DIS
LIN {X 0.133,Y -495.226,Z 679.097,A 0.000,B 0.000,C 90.000,E1 53.497} C_DIS
LIN {X 0.137,Y -476.899,Z 679.092,A 0.000,B 0.000,C 90.000,E1 52.477} C_DIS
LIN {X 0.134,Y -460.224,Z 679.086,A 0.000,B 0.000,C 90.000,E1 51.537} C_DIS
LIN {X 0.159,Y -440.422,Z 679.080,A 0.000,B 0.000,C 90.000,E1 50.356} C_DIS
LIN {X 0.114,Y -429.179,Z 679.076,A 0.000,B 0.000,C 90.000,E1 49.622} C_DIS
LIN {X 0.013,Y -428.475,Z 679.076,A 0.000,B 0.000,C 90.000,E1 49.585} C_DIS
LIN {X -0.014,Y -428.427,Z 679.076,A 0.000,B 0.000,C 90.000,E1 49.585} C_DIS
LIN {X 0.009,Y -419.592,Z 679.052,A 0.000,B 0.000,C 90.000,E1 45.364} C_DIS
LIN {X 0.083,Y -418.324,Z 679.048,A 0.000,B 0.000,C 90.000,E1 44.676} C_DIS
LIN {X 0.133,Y -414.713,Z 679.040,A 0.000,B 0.000,C 90.000,E1 43.137} C_DIS
LIN {X -0.219,Y -414.770,Z 679.026,A 0.000,B 0.000,C 90.000,E1 40.620} C_DIS
LIN {X -0.080,Y -415.426,Z 679.008,A 0.000,B 0.000,C 90.000,E1 37.523} C_DIS
LIN {X 0.122,Y -416.487,Z 678.995,A 0.000,B 0.000,C 90.000,E1 35.105} C_DIS
LIN {X -0.152,Y -417.026,Z 678.990,A 0.000,B 0.000,C 90.000,E1 34.119} C_DIS
LIN {X -0.045,Y -418.269,Z 678.976,A 0.000,B 0.000,C 90.000,E1 31.720} C_DIS
LIN {X 0.095,Y -419.202,Z 678.967,A 0.000,B 0.000,C 90.000,E1 30.001} C_DIS
LIN {X 0.017,Y -420.400,Z 678.956,A 0.000,B 0.000,C 90.000,E1 27.975} C_DIS
LIN {X 0.108,Y -421.907,Z 678.942,A 0.000,B 0.000,C 90.000,E1 25.591} C_DIS
LIN {X 0.176,Y -424.753,Z 678.924,A 0.000,B 0.000,C 90.000,E1 22.206} C_DIS
LIN {X 0.131,Y -426.672,Z 678.912,A 0.000,B 0.000,C 90.000,E1 20.194} C_DIS
LIN {X 0.130,Y -427.869,Z 678.905,A 0.000,B 0.000,C 90.000,E1 18.852} C_DIS
LIN {X 0.019,Y -429.514,Z 678.894,A 0.000,B 0.000,C 90.000,E1 16.858} C_DIS
LIN {X 0.224,Y -431.315,Z 678.883,A 0.000,B 0.000,C 90.000,E1 14.828} C_DIS
LIN {X -0.169,Y -433.344,Z 678.872,A 0.000,B 0.000,C 90.000,E1 12.883} C_DIS
LIN {X -0.184,Y -435.555,Z 678.860,A 0.000,B 0.000,C 90.000,E1 10.894} C_DIS
LIN {X 0.196,Y -438.948,Z 678.844,A 0.000,B 0.000,C 90.000,E1 7.871} C_DIS
LIN {X 0.104,Y -441.439,Z 678.833,A 0.000,B 0.000,C 90.000,E1 5.910} C_DIS
LIN {X -0.166,Y -444.988,Z 678.818,A 0.000,B 0.000,C 90.000,E1 3.326} C_DIS
LIN {X 0.105,Y -448.987,Z 678.804,A 0.000,B 0.000,C 90.000,E1 0.688} C_DIS
LIN {X 0.039,Y -451.542,Z 678.795,A 0.000,B 0.000,C 90.000,E1 359.141} C_DIS
LIN {X -0.128,Y -455.650,Z 678.783,A 0.000,B 0.000,C 90.000,E1 356.906} C_DIS
LIN {X 0.089,Y -460.480,Z 678.769,A 0.000,B 0.000,C 90.000,E1 354.318} C_DIS
LIN {X -0.189,Y -463.447,Z 678.760,A 0.000,B 0.000,C 90.000,E1 352.761} C_DIS
LIN {X -0.087,Y -467.038,Z 678.749,A 0.000,B 0.000,C 90.000,E1 350.849} C_DIS
LIN {X 0.082,Y -469.341,Z 678.742,A 0.000,B 0.000,C 90.000,E1 349.567} C_DIS
LIN {X 0.112,Y -472.132,Z 678.733,A 0.000,B 0.000,C 90.000,E1 347.993} C_DIS
LIN {X 0.122,Y -475.496,Z 678.723,A 0.000,B 0.000,C 90.000,E1 346.117} C_DIS
LIN {X 0.127,Y -480.146,Z 678.709,A 0.000,B 0.000,C 90.000,E1 343.630} C_DIS
LIN {X -0.230,Y -483.717,Z 678.699,A 0.000,B 0.000,C 90.000,E1 341.819} C_DIS
LIN {X -0.032,Y -488.091,Z 678.687,A 0.000,B 0.000,C 90.000,E1 339.645} C_DIS
LIN {X 0.064,Y -490.616,Z 678.680,A 0.000,B 0.000,C 90.000,E1 338.411} C_DIS
LIN {X -0.215,Y -493.614,Z 678.672,A 0.000,B 0.000,C 90.000,E1 336.922} C_DIS
LIN {X 0.164,Y -495.927,Z 678.665,A 0.000,B 0.000,C 90.000,E1 335.665} C_DIS
LIN {X 0.184,Y -498.991,Z 678.657,A 0.000,B 0.000,C 90.000,E1 334.152} C_DIS
LIN {X 0.070,Y -500.562,Z 678.653,A 0.000,B 0.000,C 90.000,E1 333.563} C_DIS
LIN {X -0.164,Y -502.573,Z 678.650,A 0.000,B 0.000,C 90.000,E1 332.999} C_DIS
LIN {X 0.130,Y -504.163,Z 678.648,A 0.000,B 0.000,C 90.000,E1 332.666} C_DIS
LIN {X 0.014,Y -507.347,Z 678.646,A 0.000,B 0.000,C 90.000,E1 332.231} C_DIS
LIN {X 0.022,Y -510.517,Z 678.644,A 0.000,B 0.000,C 90.000,E1 331.897} C_DIS
LIN {X -0.288,Y -519.068,Z 678.640,A 0.000,B 0.000,C 90.000,E1 331.257} C_DIS
LIN {X 0.126,Y -530.146,Z 678.636,A 0.000,B 0.000,C 90.000,E1 330.461} C_DIS
LIN {X 0.048,Y -539.294,Z 678.632,A 0.000,B 0.000,C 90.000,E1 329.822} C_DIS
LIN {X -0.349,Y -545.036,Z 678.630,A 0.000,B 0.000,C 90.000,E1 329.410} C_DIS
LIN {X -0.116,Y -552.177,Z 678.627,A 0.000,B 0.000,C 90.000,E1 328.791} C_DIS
LIN {X 0.151,Y -557.637,Z 678.624,A 0.000,B 0.000,C 90.000,E1 328.280} C_DIS
LIN {X 0.093,Y -566.848,Z 678.619,A 0.000,B 0.000,C 90.000,E1 327.406} C_DIS
LIN {X 0.233,Y -575.764,Z 678.614,A 0.000,B 0.000,C 90.000,E1 326.501} C_DIS
LIN {X 0.132,Y -585.906,Z 678.608,A 0.000,B 0.000,C 90.000,E1 325.468} C_DIS
LIN {X -0.395,Y -595.802,Z 678.603,A 0.000,B 0.000,C 90.000,E1 324.482} C_DIS
LIN {X -0.026,Y -603.782,Z 678.597,A 0.000,B 0.000,C 90.000,E1 323.543} C_DIS
LIN {X -0.013,Y -611.379,Z 678.592,A 0.000,B 0.000,C 90.000,E1 322.637} C_DIS
LIN {X 0.173,Y -615.370,Z 678.590,A 0.000,B 0.000,C 90.000,E1 322.110} C_DIS
LIN {X 0.064,Y -622.888,Z 678.584,A 0.000,B 0.000,C 90.000,E1 321.090} C_DIS
LIN {X 0.216,Y -627.221,Z 678.580,A 0.000,B 0.000,C 90.000,E1 320.436} C_DIS
LIN {X 0.276,Y -633.007,Z 678.575,A 0.000,B 0.000,C 90.000,E1 319.542} C_DIS
LIN {X -0.098,Y -639.238,Z 678.570,A 0.000,B 0.000,C 90.000,E1 318.566} C_DIS
LIN {X 0.030,Y -645.099,Z 678.564,A 0.000,B 0.000,C 90.000,E1 317.553} C_DIS
LIN {X -0.248,Y -651.275,Z 678.558,A 0.000,B 0.000,C 90.000,E1 316.458} C_DIS
LIN {X 0.052,Y -655.854,Z 678.553,A 0.000,B 0.000,C 90.000,E1 315.567} C_DIS
LIN {X -0.072,Y -660.615,Z 678.548,A 0.000,B 0.000,C 90.000,E1 314.595} C_DIS
LIN {X -0.151,Y -666.143,Z 678.541,A 0.000,B 0.000,C 90.000,E1 313.380} C_DIS
LIN {X 0.330,Y -669.381,Z 678.537,A 0.000,B 0.000,C 90.000,E1 312.609} C_DIS
LIN {X -0.074,Y -674.596,Z 678.530,A 0.000,B 0.000,C 90.000,E1 311.434} C_DIS
LIN {X 0.076,Y -678.444,Z 678.525,A 0.000,B 0.000,C 90.000,E1 310.458} C_DIS
LIN {X 0.246,Y -681.074,Z 678.521,A 0.000,B 0.000,C 90.000,E1 309.725} C_DIS
LIN {X -0.084,Y -683.484,Z 678.517,A 0.000,B 0.000,C 90.000,E1 309.036} C_DIS
LIN {X -0.248,Y -686.403,Z 678.512,A 0.000,B 0.000,C 90.000,E1 308.096} C_DIS
LIN {X -0.375,Y -688.978,Z 678.506,A 0.000,B 0.000,C 90.000,E1 307.156} C_DIS
LIN {X 0.088,Y -691.348,Z 678.501,A 0.000,B 0.000,C 90.000,E1 306.171} C_DIS
LIN {X 0.020,Y -693.415,Z 678.496,A 0.000,B 0.000,C 90.000,E1 305.231} C_DIS
LIN {X 0.146,Y -695.286,Z 678.491,A 0.000,B 0.000,C 90.000,E1 304.278} C_DIS
LIN {X -0.277,Y -696.935,Z 678.485,A 0.000,B 0.000,C 90.000,E1 303.372} C_DIS
LIN {X 0.243,Y -698.010,Z 678.481,A 0.000,B 0.000,C 90.000,E1 302.625} C_DIS
LIN {X 0.096,Y -699.579,Z 678.475,A 0.000,B 0.000,C 90.000,E1 301.465} C_DIS
LIN {X -0.323,Y -700.397,Z 678.471,A 0.000,B 0.000,C 90.000,E1 300.797} C_DIS
LIN {X -0.195,Y -701.477,Z 678.464,A 0.000,B 0.000,C 90.000,E1 299.617} C_DIS
LIN {X -0.322,Y -702.165,Z 678.459,A 0.000,B 0.000,C 90.000,E1 298.693} C_DIS
LIN {X -0.168,Y -702.996,Z 678.453,A 0.000,B 0.000,C 90.000,E1 297.513} C_DIS
LIN {X 0.017,Y -703.663,Z 678.448,A 0.000,B 0.000,C 90.000,E1 296.565} C_DIS
LIN {X -0.109,Y -704.293,Z 678.442,A 0.000,B 0.000,C 90.000,E1 295.643} C_DIS
LIN {X 0.159,Y -703.982,Z 678.440,A 0.000,B 0.000,C 90.000,E1 295.155} C_DIS
LIN {X -0.194,Y -703.684,Z 678.439,A 0.000,B 0.000,C 90.000,E1 294.951} C_DIS
LIN {X 0.078,Y -701.937,Z 678.436,A 0.000,B 0.000,C 90.000,E1 294.463} C_DIS
LIN {X 0.357,Y -700.769,Z 678.435,A 0.000,B 0.000,C 90.000,E1 294.207} C_DIS
LIN {X -0.145,Y -699.728,Z 678.434,A 0.000,B 0.000,C 90.000,E1 294.131} C_DIS
LIN {X -0.008,Y -698.477,Z 678.433,A 0.000,B 0.000,C 90.000,E1 294.003} C_DIS
LIN {X -0.254,Y -694.188,Z 678.432,A 0.000,B 0.000,C 90.000,E1 293.695} C_DIS
LIN {X 0.069,Y -692.430,Z 678.431,A 0.000,B 0.000,C 90.000,E1 293.567} C_DIS
LIN {X -0.349,Y -690.096,Z 678.431,A 0.000,B 0.000,C 90.000,E1 293.515} C_DIS
LIN {X 0.142,Y -687.273,Z 678.430,A 0.000,B 0.000,C 90.000,E1 293.387} C_DIS
LIN {X -0.116,Y -680.969,Z 678.429,A 0.000,B 0.000,C 90.000,E1 293.259} C_DIS
LIN {X 0.002,Y -678.684,Z 678.429,A 0.000,B 0.000,C 90.000,E1 293.206} C_DIS
LIN {X -0.281,Y -665.296,Z 678.428,A 0.000,B 0.000,C 90.000,E1 293.078} C_DIS
LIN {X 0.153,Y -651.639,Z 678.427,A 0.000,B 0.000,C 90.000,E1 292.845} C_DIS
LIN {X -0.297,Y -638.464,Z 678.426,A 0.000,B 0.000,C 90.000,E1 292.642} C_DIS
LIN {X 0.114,Y -628.391,Z 678.424,A 0.000,B 0.000,C 90.000,E1 292.386} C_DIS
LIN {X -0.034,Y -618.590,Z 678.423,A 0.000,B 0.000,C 90.000,E1 292.153} C_DIS
LIN {X -0.031,Y -601.516,Z 678.420,A 0.000,B 0.000,C 90.000,E1 291.663} C_DIS
LIN {X -0.168,Y -577.245,Z 678.416,A 0.000,B 0.000,C 90.000,E1 290.918} C_DIS
LIN {X 0.038,Y -562.801,Z 678.414,A 0.000,B 0.000,C 90.000,E1 290.482} C_DIS
LIN {X 0.139,Y -557.017,Z 678.412,A 0.000,B 0.000,C 90.000,E1 290.194} C_DIS
LIN {X 0.093,Y -556.945,Z 678.412,A 0.000,B 0.000,C 90.000,E1 290.194} C_DIS
LIN {X 0.341,Y -555.458,Z 678.411,A 0.000,B 0.000,C 90.000,E1 289.993} C_DIS
LIN {X 0.299,Y -555.424,Z 678.411,A 0.000,B 0.000,C 90.000,E1 289.993} C_DIS
LIN {X 0.064,Y -554.583,Z 678.410,A 0.000,B 0.000,C 90.000,E1 289.704} C_DIS
LIN {X -0.190,Y -554.210,Z 678.406,A 0.000,B 0.000,C 90.000,E1 289.033} C_DIS
LIN {X 0.229,Y -553.964,Z 678.399,A 0.000,B 0.000,C 90.000,E1 287.873} C_DIS
LIN {X -0.105,Y -553.378,Z 678.389,A 0.000,B 0.000,C 90.000,E1 285.953} C_DIS
LIN {X 0.203,Y -552.737,Z 678.379,A 0.000,B 0.000,C 90.000,E1 284.245} C_DIS
LIN {X -0.149,Y -552.029,Z 678.372,A 0.000,B 0.000,C 90.000,E1 282.883} C_DIS
LIN {X -0.102,Y -551.351,Z 678.364,A 0.000,B 0.000,C 90.000,E1 281.478} C_DIS
LIN {X 0.170,Y -550.317,Z 678.351,A 0.000,B 0.000,C 90.000,E1 279.208} C_DIS
LIN {X -0.189,Y -549.622,Z 678.337,A 0.000,B 0.000,C 90.000,E1 276.720} C_DIS
LIN {X 0.224,Y -549.381,Z 678.328,A 0.000,B 0.000,C 90.000,E1 274.992} C_DIS
LIN {X 0.038,Y -549.245,Z 678.319,A 0.000,B 0.000,C 90.000,E1 273.326} C_DIS
LIN {X -0.228,Y -549.000,Z 678.311,A 0.000,B 0.000,C 90.000,E1 271.949} C_DIS
LIN {X 0.043,Y -548.436,Z 678.303,A 0.000,B 0.000,C 90.000,E1 270.516} C_DIS
LIN {X 0.243,Y -547.790,Z 678.297,A 0.000,B 0.000,C 90.000,E1 269.370} C_DIS
LIN {X 0.031,Y -546.654,Z 678.286,A 0.000,B 0.000,C 90.000,E1 267.421} C_DIS
LIN {X 0.218,Y -545.963,Z 678.279,A 0.000,B 0.000,C 90.000,E1 266.274} C_DIS
LIN {X -0.080,Y -544.886,Z 678.272,A 0.000,B 0.000,C 90.000,E1 264.894} C_DIS
LIN {X 0.123,Y -544.024,Z 678.265,A 0.000,B 0.000,C 90.000,E1 263.742} C_DIS
LIN {X -0.230,Y -542.906,Z 678.259,A 0.000,B 0.000,C 90.000,E1 262.648} C_DIS
LIN {X 0.151,Y -540.803,Z 678.248,A 0.000,B 0.000,C 90.000,E1 260.622} C_DIS
LIN {X 0.207,Y -538.731,Z 678.235,A 0.000,B 0.000,C 90.000,E1 258.342} C_DIS
LIN {X 0.143,Y -537.072,Z 678.224,A 0.000,B 0.000,C 90.000,E1 256.353} C_DIS
LIN {X 0.039,Y -535.862,Z 678.216,A 0.000,B 0.000,C 90.000,E1 254.936} C_DIS
LIN {X 0.008,Y -534.705,Z 678.210,A 0.000,B 0.000,C 90.000,E1 253.795} C_DIS
LIN {X 0.200,Y -532.947,Z 678.201,A 0.000,B 0.000,C 90.000,E1 252.054} C_DIS
LIN {X -0.159,Y -531.267,Z 678.191,A 0.000,B 0.000,C 90.000,E1 250.369} C_DIS
LIN {X -0.080,Y -529.859,Z 678.185,A 0.000,B 0.000,C 90.000,E1 249.209} C_DIS
LIN {X 0.172,Y -528.300,Z 678.178,A 0.000,B 0.000,C 90.000,E1 248.028} C_DIS
LIN {X 0.061,Y -525.775,Z 678.168,A 0.000,B 0.000,C 90.000,E1 246.305} C_DIS
LIN {X -0.166,Y -522.839,Z 678.159,A 0.000,B 0.000,C 90.000,E1 244.588} C_DIS
LIN {X 0.050,Y -521.284,Z 678.154,A 0.000,B 0.000,C 90.000,E1 243.691} C_DIS
LIN {X -0.032,Y -517.826,Z 678.144,A 0.000,B 0.000,C 90.000,E1 241.948} C_DIS
LIN {X -0.217,Y -515.484,Z 678.138,A 0.000,B 0.000,C 90.000,E1 240.795} C_DIS
LIN {X -0.293,Y -511.078,Z 678.126,A 0.000,B 0.000,C 90.000,E1 238.742} C_DIS
LIN {X 0.150,Y -507.132,Z 678.116,A 0.000,B 0.000,C 90.000,E1 236.914} C_DIS
LIN {X 0.069,Y -502.973,Z 678.106,A 0.000,B 0.000,C 90.000,E1 235.135} C_DIS
LIN {X 0.186,Y -499.289,Z 678.098,A 0.000,B 0.000,C 90.000,E1 233.623} C_DIS
LIN {X 0.246,Y -495.607,Z 678.090,A 0.000,B 0.000,C 90.000,E1 232.110} C_DIS
LIN {X 0.235,Y -490.468,Z 678.078,A 0.000,B 0.000,C 90.000,E1 229.989} C_DIS
LIN {X 0.050,Y -486.846,Z 678.069,A 0.000,B 0.000,C 90.000,E1 228.485} C_DIS
LIN {X 0.117,Y -483.208,Z 678.061,A 0.000,B 0.000,C 90.000,E1 226.944} C_DIS
LIN {X 0.221,Y -478.882,Z 678.051,A 0.000,B 0.000,C 90.000,E1 225.081} C_DIS
LIN {X 0.123,Y -475.214,Z 678.042,A 0.000,B 0.000,C 90.000,E1 223.542} C_DIS
LIN {X 0.063,Y -470.980,Z 678.032,A 0.000,B 0.000,C 90.000,E1 221.676} C_DIS
LIN {X -0.046,Y -466.934,Z 678.021,A 0.000,B 0.000,C 90.000,E1 219.806} C_DIS
LIN {X -0.129,Y -462.307,Z 678.009,A 0.000,B 0.000,C 90.000,E1 217.604} C_DIS
LIN {X 0.016,Y -457.865,Z 677.997,A 0.000,B 0.000,C 90.000,E1 215.358} C_DIS
LIN {X -0.202,Y -455.006,Z 677.988,A 0.000,B 0.000,C 90.000,E1 213.785} C_DIS
LIN {X 0.247,Y -451.287,Z 677.977,A 0.000,B 0.000,C 90.000,E1 211.799} C_DIS
LIN {X 0.207,Y -447.022,Z 677.964,A 0.000,B 0.000,C 90.000,E1 209.539} C_DIS
LIN {X 0.169,Y -443.459,Z 677.953,A 0.000,B 0.000,C 90.000,E1 207.590} C_DIS
LIN {X 0.004,Y -440.560,Z 677.944,A 0.000,B 0.000,C 90.000,E1 205.976} C_DIS
LIN {X -0.013,Y -437.531,Z 677.935,A 0.000,B 0.000,C 90.000,E1 204.335} C_DIS
LIN {X -0.095,Y -435.201,Z 677.928,A 0.000,B 0.000,C 90.000,E1 203.025} C_DIS
LIN {X 0.011,Y -432.191,Z 677.919,A 0.000,B 0.000,C 90.000,E1 201.354} C_DIS
LIN {X 0.116,Y -428.545,Z 677.908,A 0.000,B 0.000,C 90.000,E1 199.341} C_DIS
LIN {X 0.122,Y -424.996,Z 677.896,A 0.000,B 0.000,C 90.000,E1 197.330} C_DIS
LIN {X 0.071,Y -421.624,Z 677.885,A 0.000,B 0.000,C 90.000,E1 195.315} C_DIS
LIN {X -0.112,Y -418.689,Z 677.876,A 0.000,B 0.000,C 90.000,E1 193.647} C_DIS
LIN {X 0.134,Y -413.645,Z 677.859,A 0.000,B 0.000,C 90.000,E1 190.546} C_DIS
LIN {X -0.038,Y -410.430,Z 677.847,A 0.000,B 0.000,C 90.000,E1 188.511} C_DIS
LIN {X 0.053,Y -407.274,Z 677.836,A 0.000,B 0.000,C 90.000,E1 186.429} C_DIS
LIN {X -0.096,Y -403.085,Z 677.818,A 0.000,B 0.000,C 90.000,E1 183.326} C_DIS
LIN {X 0.065,Y -400.194,Z 677.805,A 0.000,B 0.000,C 90.000,E1 180.859} C_DIS
LIN {X 0.122,Y -397.830,Z 677.791,A 0.000,B 0.000,C 90.000,E1 178.396} C_DIS
LIN {X 0.019,Y -395.380,Z 677.774,A 0.000,B 0.000,C 90.000,E1 175.241} C_DIS
LIN {X 0.025,Y -393.914,Z 677.758,A 0.000,B 0.000,C 90.000,E1 172.413} C_DIS
LIN {X 0.040,Y -392.985,Z 677.742,A 0.000,B 0.000,C 90.000,E1 169.577} C_DIS
LIN {X -0.112,Y -392.608,Z 677.728,A 0.000,B 0.000,C 90.000,E1 167.117} C_DIS
LIN {X -0.096,Y -392.287,Z 677.711,A 0.000,B 0.000,C 90.000,E1 163.921} C_DIS
LIN {X 0.138,Y -392.304,Z 677.697,A 0.000,B 0.000,C 90.000,E1 161.402} C_DIS
LIN {X 0.017,Y -392.438,Z 677.687,A 0.000,B 0.000,C 90.000,E1 159.645} C_DIS
LIN {X -0.139,Y -392.690,Z 677.675,A 0.000,B 0.000,C 90.000,E1 157.539} C_DIS
LIN {X -0.090,Y -392.940,Z 677.661,A 0.000,B 0.000,C 90.000,E1 155.049} C_DIS
LIN {X -0.094,Y -393.341,Z 677.650,A 0.000,B 0.000,C 90.000,E1 152.922} C_DIS
LIN {X -0.085,Y -393.792,Z 677.638,A 0.000,B 0.000,C 90.000,E1 150.795} C_DIS
LIN {X -0.027,Y -394.280,Z 677.626,A 0.000,B 0.000,C 90.000,E1 148.663} C_DIS
LIN {X 0.198,Y -395.369,Z 677.610,A 0.000,B 0.000,C 90.000,E1 145.801} C_DIS
LIN {X 0.118,Y -397.074,Z 677.593,A 0.000,B 0.000,C 90.000,E1 142.637} C_DIS
LIN {X -0.021,Y -398.709,Z 677.579,A 0.000,B 0.000,C 90.000,E1 140.194} C_DIS
LIN {X 0.145,Y -400.666,Z 677.565,A 0.000,B 0.000,C 90.000,E1 137.715} C_DIS
LIN {X -0.038,Y -403.340,Z 677.548,A 0.000,B 0.000,C 90.000,E1 134.595} C_DIS
LIN {X 0.103,Y -404.704,Z 677.543,A 0.000,B 0.000,C 90.000,E1 133.704} C_DIS
LIN {X -0.177,Y -406.574,Z 677.539,A 0.000,B 0.000,C 90.000,E1 133.014} C_DIS
LIN {X 0.234,Y -408.261,Z 677.537,A 0.000,B 0.000,C 90.000,E1 132.609} C_DIS
LIN {X 0.154,Y -408.962,Z 677.536,A 0.000,B 0.000,C 90.000,E1 132.447} C_DIS
LIN {X 0.074,Y -410.125,Z 677.535,A 0.000,B 0.000,C 90.000,E1 132.285} C_DIS
LIN {X 0.228,Y -412.574,Z 677.533,A 0.000,B 0.000,C 90.000,E1 131.919} C_DIS
LIN {X -0.015,Y -417.671,Z 677.530,A 0.000,B 0.000,C 90.000,E1 131.434} C_DIS
LIN {X -0.079,Y -429.202,Z 677.525,A 0.000,B 0.000,C 90.000,E1 130.458} C_DIS
LIN {X -0.082,Y -447.966,Z 677.516,A 0.000,B 0.000,C 90.000,E1 128.955} C_DIS
LIN {X -0.066,Y -463.666,Z 677.510,A 0.000,B 0.000,C 90.000,E1 127.729} C_DIS
LIN {X 0.252,Y -471.161,Z 677.506,A 0.000,B 0.000,C 90.000,E1 127.076} C_DIS
LIN {X -0.267,Y -480.132,Z 677.502,A 0.000,B 0.000,C 90.000,E1 126.377} C_DIS
LIN {X 0.211,Y -485.938,Z 677.499,A 0.000,B 0.000,C 90.000,E1 125.804} C_DIS
LIN {X -0.031,Y -490.237,Z 677.497,A 0.000,B 0.000,C 90.000,E1 125.438} C_DIS
LIN {X -0.119,Y -499.867,Z 677.492,A 0.000,B 0.000,C 90.000,E1 124.532} C_DIS
LIN {X -0.087,Y -505.208,Z 677.489,A 0.000,B 0.000,C 90.000,E1 123.992} C_DIS
LIN {X -0.093,Y -511.968,Z 677.485,A 0.000,B 0.000,C 90.000,E1 123.293} C_DIS
LIN {X -0.086,Y -518.146,Z 677.481,A 0.000,B 0.000,C 90.000,E1 122.625} C_DIS
LIN {X 0.138,Y -524.176,Z 677.477,A 0.000,B 0.000,C 90.000,E1 121.878} C_DIS
LIN {X 0.086,Y -526.638,Z 677.476,A 0.000,B 0.000,C 90.000,E1 121.592} C_DIS
LIN {X 0.181,Y -530.999,Z 677.472,A 0.000,B 0.000,C 90.000,E1 121.003} C_DIS
LIN {X -0.295,Y -535.950,Z 677.468,A 0.000,B 0.000,C 90.000,E1 120.335} C_DIS
LIN {X -0.128,Y -539.464,Z 677.465,A 0.000,B 0.000,C 90.000,E1 119.745} C_DIS
LIN {X -0.064,Y -543.458,Z 677.461,A 0.000,B 0.000,C 90.000,E1 119.027} C_DIS
LIN {X -0.284,Y -547.041,Z 677.457,A 0.000,B 0.000,C 90.000,E1 118.359} C_DIS
LIN {X 0.097,Y -551.585,Z 677.452,A 0.000,B 0.000,C 90.000,E1 117.334} C_DIS
LIN {X -0.111,Y -554.052,Z 677.449,A 0.000,B 0.000,C 90.000,E1 116.796} C_DIS
LIN {X 0.007,Y -558.487,Z 677.443,A 0.000,B 0.000,C 90.000,E1 115.668} C_DIS
LIN {X 0.126,Y -561.660,Z 677.438,A 0.000,B 0.000,C 90.000,E1 114.823} C_DIS
LIN {X -0.193,Y -564.523,Z 677.433,A 0.000,B 0.000,C 90.000,E1 114.027} C_DIS
LIN {X -0.249,Y -567.089,Z 677.429,A 0.000,B 0.000,C 90.000,E1 113.206} C_DIS
LIN {X 0.058,Y -569.974,Z 677.423,A 0.000,B 0.000,C 90.000,E1 112.078} C_DIS
LIN {X 0.014,Y -571.358,Z 677.420,A 0.000,B 0.000,C 90.000,E1 111.535} C_DIS
LIN {X 0.170,Y -573.639,Z 677.414,A 0.000,B 0.000,C 90.000,E1 110.429} C_DIS
LIN {X 0.162,Y -575.855,Z 677.408,A 0.000,B 0.000,C 90.000,E1 109.341} C_DIS
LIN {X -0.334,Y -578.957,Z 677.399,A 0.000,B 0.000,C 90.000,E1 107.764} C_DIS
LIN {X -0.055,Y -581.558,Z 677.391,A 0.000,B 0.000,C 90.000,E1 106.386} C_DIS
LIN {X 0.267,Y -584.073,Z 677.384,A 0.000,B 0.000,C 90.000,E1 105.009} C_DIS
LIN {X 0.149,Y -586.934,Z 677.375,A 0.000,B 0.000,C 90.000,E1 103.411} C_DIS
LIN {X 0.212,Y -590.199,Z 677.364,A 0.000,B 0.000,C 90.000,E1 101.535} C_DIS
LIN {X 0.238,Y -593.467,Z 677.354,A 0.000,B 0.000,C 90.000,E1 99.670} C_DIS
LIN {X -0.042,Y -596.036,Z 677.345,A 0.000,B 0.000,C 90.000,E1 98.106} C_DIS
LIN {X 0.035,Y -597.979,Z 677.338,A 0.000,B 0.000,C 90.000,E1 96.777} C_DIS
LIN {X 0.080,Y -599.846,Z 677.330,A 0.000,B 0.000,C 90.000,E1 95.454} C_DIS
LIN {X 0.285,Y -600.919,Z 677.326,A 0.000,B 0.000,C 90.000,E1 94.645} C_DIS
LIN {X 0.018,Y -602.857,Z 677.317,A 0.000,B 0.000,C 90.000,E1 93.094} C_DIS
LIN {X 0.099,Y -604.150,Z 677.310,A 0.000,B 0.000,C 90.000,E1 91.776} C_DIS
LIN {X -0.073,Y -605.037,Z 677.304,A 0.000,B 0.000,C 90.000,E1 90.745} C_DIS
LIN {X 0.302,Y -605.991,Z 677.295,A 0.000,B 0.000,C 90.000,E1 89.141} C_DIS
LIN {X 0.173,Y -606.350,Z 677.290,A 0.000,B 0.000,C 90.000,E1 88.108} C_DIS
LIN {X -0.282,Y -606.703,Z 677.282,A 0.000,B 0.000,C 90.000,E1 86.846} C_DIS
LIN {X 0.211,Y -606.775,Z 677.277,A 0.000,B 0.000,C 90.000,E1 85.755} C_DIS
LIN {X -0.199,Y -606.698,Z 677.269,A 0.000,B 0.000,C 90.000,E1 84.489} C_DIS
LIN {X 0.024,Y -606.554,Z 677.265,A 0.000,B 0.000,C 90.000,E1 83.685} C_DIS
LIN {X 0.274,Y -606.096,Z 677.258,A 0.000,B 0.000,C 90.000,E1 82.356} C_DIS
LIN {X 0.190,Y -605.612,Z 677.252,A 0.000,B 0.000,C 90.000,E1 81.319} C_DIS
LIN {X 0.187,Y -604.784,Z 677.246,A 0.000,B 0.000,C 90.000,E1 80.274} C_DIS
LIN {X 0.212,Y -603.252,Z 677.237,A 0.000,B 0.000,C 90.000,E1 78.701} C_DIS
LIN {X -0.298,Y -602.126,Z 677.232,A 0.000,B 0.000,C 90.000,E1 77.701} C_DIS
LIN {X 0.074,Y -600.510,Z 677.224,A 0.000,B 0.000,C 90.000,E1 76.353} C_DIS
LIN {X 0.262,Y -599.153,Z 677.218,A 0.000,B 0.000,C 90.000,E1 75.283} C_DIS
LIN {X -0.141,Y -597.678,Z 677.213,A 0.000,B 0.000,C 90.000,E1 74.267} C_DIS
LIN {X -0.281,Y -595.702,Z 677.205,A 0.000,B 0.000,C 90.000,E1 72.960} C_DIS
LIN {X 0.017,Y -593.989,Z 677.199,A 0.000,B 0.000,C 90.000,E1 71.873} C_DIS
LIN {X 0.293,Y -592.151,Z 677.193,A 0.000,B 0.000,C 90.000,E1 70.786} C_DIS
LIN {X -0.019,Y -590.174,Z 677.188,A 0.000,B 0.000,C 90.000,E1 69.752} C_DIS
LIN {X 0.186,Y -587.944,Z 677.182,A 0.000,B 0.000,C 90.000,E1 68.666} C_DIS
LIN {X -0.179,Y -586.155,Z 677.177,A 0.000,B 0.000,C 90.000,E1 67.901} C_DIS
LIN {X 0.178,Y -583.374,Z 677.171,A 0.000,B 0.000,C 90.000,E1 66.794} C_DIS
LIN {X 0.085,Y -581.097,Z 677.167,A 0.000,B 0.000,C 90.000,E1 65.997} C_DIS
LIN {X 0.059,Y -577.809,Z 677.161,A 0.000,B 0.000,C 90.000,E1 64.921} C_DIS
LIN {X 0.139,Y -575.071,Z 677.156,A 0.000,B 0.000,C 90.000,E1 64.101} C_DIS
LIN {X -0.067,Y -572.160,Z 677.152,A 0.000,B 0.000,C 90.000,E1 63.307} C_DIS
LIN {X 0.119,Y -570.178,Z 677.149,A 0.000,B 0.000,C 90.000,E1 62.743} C_DIS
LIN {X -0.125,Y -566.979,Z 677.144,A 0.000,B 0.000,C 90.000,E1 61.948} C_DIS
LIN {X 0.008,Y -562.801,Z 677.139,A 0.000,B 0.000,C 90.000,E1 60.973} C_DIS
LIN {X 0.107,Y -560.242,Z 677.136,A 0.000,B 0.000,C 90.000,E1 60.411} C_DIS
LIN {X -0.133,Y -556.637,Z 677.132,A 0.000,B 0.000,C 90.000,E1 59.744} C_DIS
LIN {X 0.357,Y -552.522,Z 677.128,A 0.000,B 0.000,C 90.000,E1 58.997} C_DIS
LIN {X 0.174,Y -548.969,Z 677.125,A 0.000,B 0.000,C 90.000,E1 58.456} C_DIS
LIN {X 0.011,Y -545.124,Z 677.122,A 0.000,B 0.000,C 90.000,E1 57.916} C_DIS
LIN {X 0.004,Y -540.036,Z 677.118,A 0.000,B 0.000,C 90.000,E1 57.248} C_DIS
LIN {X 0.013,Y -535.482,Z 677.115,A 0.000,B 0.000,C 90.000,E1 56.707} C_DIS
LIN {X 0.132,Y -530.319,Z 677.112,A 0.000,B 0.000,C 90.000,E1 56.167} C_DIS
LIN {X -0.184,Y -526.130,Z 677.110,A 0.000,B 0.000,C 90.000,E1 55.801} C_DIS
LIN {X -0.101,Y -520.108,Z 677.107,A 0.000,B 0.000,C 90.000,E1 55.308} C_DIS
LIN {X -0.024,Y -513.947,Z 677.105,A 0.000,B 0.000,C 90.000,E1 54.848} C_DIS
LIN {X -0.095,Y -509.166,Z 677.103,A 0.000,B 0.000,C 90.000,E1 54.529} C_DIS
LIN {X -0.109,Y -502.417,Z 677.101,A 0.000,B 0.000,C 90.000,E1 54.116} C_DIS
LIN {X 0.092,Y -495.688,Z 677.098,A 0.000,B 0.000,C 90.000,E1 53.703} C_DIS
LIN {X -0.048,Y -485.822,Z 677.095,A 0.000,B 0.000,C 90.000,E1 53.176} C_DIS
LIN {X -0.254,Y -469.204,Z 677.090,A 0.000,B 0.000,C 90.000,E1 52.271} C_DIS
LIN {X -0.183,Y -442.578,Z 677.082,A 0.000,B 0.000,C 90.000,E1 50.723} C_DIS
LIN {X -0.072,Y -429.016,Z 677.077,A 0.000,B 0.000,C 90.000,E1 49.828} C_DIS
LIN {X -0.094,Y -428.993,Z 677.077,A 0.000,B 0.000,C 90.000,E1 49.828} C_DIS
LIN {X -0.109,Y -420.073,Z 677.054,A 0.000,B 0.000,C 90.000,E1 45.648} C_DIS
LIN {X -0.031,Y -418.875,Z 677.050,A 0.000,B 0.000,C 90.000,E1 44.960} C_DIS
LIN {X 0.040,Y -417.319,Z 677.046,A 0.000,B 0.000,C 90.000,E1 44.271} C_DIS
LIN {X 0.011,Y -415.129,Z 677.041,A 0.000,B 0.000,C 90.000,E1 43.338} C_DIS
LIN {X -0.079,Y -415.224,Z 677.027,A 0.000,B 0.000,C 90.000,E1 40.782} C_DIS
LIN {X -0.064,Y -415.988,Z 677.008,A 0.000,B 0.000,C 90.000,E1 37.363} C_DIS
LIN {X 0.092,Y -417.308,Z 676.992,A 0.000,B 0.000,C 90.000,E1 34.612} C_DIS
LIN {X 0.170,Y -418.702,Z 676.977,A 0.000,B 0.000,C 90.000,E1 31.878} C_DIS
LIN {X -0.035,Y -419.638,Z 676.968,A 0.000,B 0.000,C 90.000,E1 30.207} C_DIS
LIN {X -0.137,Y -421.007,Z 676.955,A 0.000,B 0.000,C 90.000,E1 27.847} C_DIS
LIN {X -0.030,Y -422.531,Z 676.941,A 0.000,B 0.000,C 90.000,E1 25.463} C_DIS
LIN {X 0.061,Y -425.404,Z 676.923,A 0.000,B 0.000,C 90.000,E1 22.078} C_DIS
LIN {X 0.027,Y -427.324,Z 676.912,A 0.000,B 0.000,C 90.000,E1 20.066} C_DIS
LIN {X -0.166,Y -428.738,Z 676.902,A 0.000,B 0.000,C 90.000,E1 18.417} C_DIS
LIN {X -0.069,Y -430.068,Z 676.893,A 0.000,B 0.000,C 90.000,E1 16.732} C_DIS
LIN {X -0.071,Y -431.546,Z 676.884,A 0.000,B 0.000,C 90.000,E1 15.064} C_DIS
LIN {X 0.082,Y -433.835,Z 676.871,A 0.000,B 0.000,C 90.000,E1 12.715} C_DIS
LIN {X 0.089,Y -435.999,Z 676.860,A 0.000,B 0.000,C 90.000,E1 10.725} C_DIS
LIN {X -0.082,Y -438.970,Z 676.845,A 0.000,B 0.000,C 90.000,E1 8.106} C_DIS
LIN {X 0.167,Y -441.038,Z 676.836,A 0.000,B 0.000,C 90.000,E1 6.429} C_DIS
LIN {X 0.203,Y -444.036,Z 676.823,A 0.000,B 0.000,C 90.000,E1 4.131} C_DIS
LIN {X 0.164,Y -446.872,Z 676.812,A 0.000,B 0.000,C 90.000,E1 2.178} C_DIS
LIN {X 0.171,Y -450.684,Z 676.799,A 0.000,B 0.000,C 90.000,E1 359.771} C_DIS
LIN {X -0.123,Y -455.809,Z 676.783,A 0.000,B 0.000,C 90.000,E1 356.906} C_DIS
LIN {X -0.130,Y -459.995,Z 676.770,A 0.000,B 0.000,C 90.000,E1 354.666} C_DIS
LIN {X -0.175,Y -463.577,Z 676.760,A 0.000,B 0.000,C 90.000,E1 352.761} C_DIS
LIN {X -0.070,Y -467.142,Z 676.749,A 0.000,B 0.000,C 90.000,E1 350.849} C_DIS
LIN {X 0.016,Y -469.444,Z 676.742,A 0.000,B 0.000,C 90.000,E1 349.577} C_DIS
LIN {X 0.133,Y -472.238,Z 676.733,A 0.000,B 0.000,C 90.000,E1 347.993} C_DIS
LIN {X -0.020,Y -476.175,Z 676.721,A 0.000,B 0.000,C 90.000,E1 345.825} C_DIS
LIN {X 0.154,Y -480.250,Z 676.709,A 0.000,B 0.000,C 90.000,E1 343.630} C_DIS
LIN {X -0.201,Y -483.816,Z 676.699,A 0.000,B 0.000,C 90.000,E1 341.819} C_DIS
LIN {X 0.000,Y -488.182,Z 676.687,A 0.000,B 0.000,C 90.000,E1 339.645} C_DIS
LIN {X 0.128,Y -491.294,Z 676.678,A 0.000,B 0.000,C 90.000,E1 338.103} C_DIS
LIN {X -0.138,Y -494.273,Z 676.670,A 0.000,B 0.000,C 90.000,E1 336.613} C_DIS
LIN {X -0.151,Y -497.110,Z 676.662,A 0.000,B 0.000,C 90.000,E1 335.101} C_DIS
LIN {X -0.172,Y -499.587,Z 676.655,A 0.000,B 0.000,C 90.000,E1 333.896} C_DIS
LIN {X 0.167,Y -501.159,Z 676.652,A 0.000,B 0.000,C 90.000,E1 333.256} C_DIS
LIN {X 0.035,Y -502.647,Z 676.649,A 0.000,B 0.000,C 90.000,E1 332.820} C_DIS
LIN {X -0.104,Y -504.945,Z 676.646,A 0.000,B 0.000,C 90.000,E1 332.359} C_DIS
LIN {X 0.204,Y -506.997,Z 676.645,A 0.000,B 0.000,C 90.000,E1 332.025} C_DIS
LIN {X 0.062,Y -511.093,Z 676.642,A 0.000,B 0.000,C 90.000,E1 331.591} C_DIS
LIN {X -0.249,Y -515.496,Z 676.640,A 0.000,B 0.000,C 90.000,E1 331.257} C_DIS
LIN {X 0.141,Y -524.309,Z 676.637,A 0.000,B 0.000,C 90.000,E1 330.589} C_DIS
LIN {X -0.292,Y -533.592,Z 676.633,A 0.000,B 0.000,C 90.000,E1 329.999} C_DIS
LIN {X -0.241,Y -538.175,Z 676.631,A 0.000,B 0.000,C 90.000,E1 329.665} C_DIS
LIN {X 0.023,Y -546.906,Z 676.628,A 0.000,B 0.000,C 90.000,E1 328.948} C_DIS
LIN {X 0.254,Y -553.974,Z 676.624,A 0.000,B 0.000,C 90.000,E1 328.329} C_DIS
LIN {X 0.290,Y -563.427,Z 676.619,A 0.000,B 0.000,C 90.000,E1 327.454} C_DIS
LIN {X 0.316,Y -573.870,Z 676.614,A 0.000,B 0.000,C 90.000,E1 326.421} C_DIS
LIN {X 0.220,Y -585.366,Z 676.607,A 0.000,B 0.000,C 90.000,E1 325.261} C_DIS
LIN {X 0.150,Y -594.142,Z 676.602,A 0.000,B 0.000,C 90.000,E1 324.356} C_DIS
LIN {X 0.326,Y -602.445,Z 676.597,A 0.000,B 0.000,C 90.000,E1 323.417} C_DIS
LIN {X -0.276,Y -610.276,Z 676.592,A 0.000,B 0.000,C 90.000,E1 322.557} C_DIS
LIN {X -0.235,Y -615.373,Z 676.588,A 0.000,B 0.000,C 90.000,E1 321.904} C_DIS
LIN {X 0.166,Y -622.025,Z 676.583,A 0.000,B 0.000,C 90.000,E1 320.964} C_DIS
LIN {X 0.339,Y -625.561,Z 676.580,A 0.000,B 0.000,C 90.000,E1 320.436} C_DIS
LIN {X -0.099,Y -631.495,Z 676.576,A 0.000,B 0.000,C 90.000,E1 319.585} C_DIS
LIN {X -0.011,Y -637.830,Z 676.570,A 0.000,B 0.000,C 90.000,E1 318.566} C_DIS
LIN {X -0.396,Y -644.521,Z 676.564,A 0.000,B 0.000,C 90.000,E1 317.472} C_DIS
LIN {X -0.197,Y -650.082,Z 676.558,A 0.000,B 0.000,C 90.000,E1 316.458} C_DIS
LIN {X 0.088,Y -654.739,Z 676.553,A 0.000,B 0.000,C 90.000,E1 315.567} C_DIS
LIN {X -0.034,Y -659.013,Z 676.548,A 0.000,B 0.000,C 90.000,E1 314.717} C_DIS
LIN {X -0.109,Y -663.074,Z 676.544,A 0.000,B 0.000,C 90.000,E1 313.866} C_DIS
LIN {X 0.336,Y -667.534,Z 676.538,A 0.000,B 0.000,C 90.000,E1 312.852} C_DIS
LIN {X -0.093,Y -672.909,Z 676.532,A 0.000,B 0.000,C 90.000,E1 311.676} C_DIS
LIN {X 0.037,Y -676.857,Z 676.526,A 0.000,B 0.000,C 90.000,E1 310.701} C_DIS
LIN {X -0.327,Y -679.670,Z 676.522,A 0.000,B 0.000,C 90.000,E1 310.011} C_DIS
LIN {X -0.145,Y -682.221,Z 676.518,A 0.000,B 0.000,C 90.000,E1 309.277} C_DIS
LIN {X -0.283,Y -685.930,Z 676.512,A 0.000,B 0.000,C 90.000,E1 308.096} C_DIS
LIN {X -0.415,Y -688.563,Z 676.506,A 0.000,B 0.000,C 90.000,E1 307.156} C_DIS
LIN {X 0.041,Y -690.971,Z 676.501,A 0.000,B 0.000,C 90.000,E1 306.171} C_DIS
LIN {X -0.031,Y -693.108,Z 676.496,A 0.000,B 0.000,C 90.000,E1 305.231} C_DIS
LIN {X 0.091,Y -695.020,Z 676.491,A 0.000,B 0.000,C 90.000,E1 304.278} C_DIS
LIN {X -0.334,Y -696.730,Z 676.485,A 0.000,B 0.000,C 90.000,E1 303.372} C_DIS
LIN {X 0.182,Y -697.847,Z 676.481,A 0.000,B 0.000,C 90.000,E1 302.625} C_DIS
LIN {X 0.033,Y -699.479,Z 676.475,A 0.000,B 0.000,C 90.000,E1 301.465} C_DIS
LIN {X -0.122,Y -700.559,Z 676.470,A 0.000,B 0.000,C 90.000,E1 300.541} C_DIS
LIN {X 0.087,Y -701.465,Z 676.464,A 0.000,B 0.000,C 90.000,E1 299.589} C_DIS
LIN {X -0.387,Y -702.186,Z 676.459,A 0.000,B 0.000,C 90.000,E1 298.693} C_DIS
LIN {X 0.110,Y -702.898,Z 676.454,A 0.000,B 0.000,C 90.000,E1 297.719} C_DIS
LIN {X -0.046,Y -703.749,Z 676.448,A 0.000,B 0.000,C 90.000,E1 296.565} C_DIS
LIN {X -0.171,Y -704.378,Z 676.442,A 0.000,B 0.000,C 90.000,E1 295.643} C_DIS
LIN {X 0.097,Y -704.054,Z 676.440,A 0.000,B 0.000,C 90.000,E1 295.155} C_DIS
LIN {X -0.255,Y -703.716,Z 676.439,A 0.000,B 0.000,C 90.000,E1 294.951} C_DIS
LIN {X 0.017,Y -701.911,Z 676.436,A 0.000,B 0.000,C 90.000,E1 294.463} C_DIS
LIN {X 0.295,Y -700.686,Z 676.435,A 0.000,B 0.000,C 90.000,E1 294.207} C_DIS
LIN {X -0.206,Y -699.621,Z 676.434,A 0.000,B 0.000,C 90.000,E1 294.131} C_DIS
LIN {X -0.078,Y -693.961,Z 676.432,A 0.000,B 0.000,C 90.000,E1 293.695} C_DIS
LIN {X -0.033,Y -692.238,Z 676.431,A 0.000,B 0.000,C 90.000,E1 293.590} C_DIS
LIN {X -0.188,Y -689.844,Z 676.431,A 0.000,B 0.000,C 90.000,E1 293.515} C_DIS
LIN {X -0.319,Y -684.730,Z 676.430,A 0.000,B 0.000,C 90.000,E1 293.387} C_DIS
LIN {X 0.086,Y -680.840,Z 676.429,A 0.000,B 0.000,C 90.000,E1 293.259} C_DIS
LIN {X 0.195,Y -678.315,Z 676.429,A 0.000,B 0.000,C 90.000,E1 293.206} C_DIS
LIN {X -0.040,Y -665.104,Z 676.428,A 0.000,B 0.000,C 90.000,E1 293.078} C_DIS
LIN {X -0.234,Y -651.501,Z 676.427,A 0.000,B 0.000,C 90.000,E1 292.898} C_DIS
LIN {X -0.093,Y -638.333,Z 676.426,A 0.000,B 0.000,C 90.000,E1 292.642} C_DIS
LIN {X 0.073,Y -628.281,Z 676.425,A 0.000,B 0.000,C 90.000,E1 292.408} C_DIS
LIN {X 0.157,Y -618.468,Z 676.423,A 0.000,B 0.000,C 90.000,E1 292.153} C_DIS
LIN {X 0.154,Y -601.424,Z 676.420,A 0.000,B 0.000,C 90.000,E1 291.663} C_DIS
LIN {X -0.051,Y -577.049,Z 676.416,A 0.000,B 0.000,C 90.000,E1 290.918} C_DIS
LIN {X 0.158,Y -562.690,Z 676.414,A 0.000,B 0.000,C 90.000,E1 290.482} C_DIS
LIN {X -0.238,Y -557.089,Z 676.412,A 0.000,B 0.000,C 90.000,E1 290.248} C_DIS
LIN {X -0.288,Y -556.995,Z 676.412,A 0.000,B 0.000,C 90.000,E1 290.248} C_DIS
LIN {X 0.349,Y -555.391,Z 676.411,A 0.000,B 0.000,C 90.000,E1 289.993} C_DIS
LIN {X 0.306,Y -555.370,Z 676.411,A 0.000,B 0.000,C 90.000,E1 289.993} C_DIS
LIN {X -0.055,Y -554.571,Z 676.409,A 0.000,B 0.000,C 90.000,E1 289.704} C_DIS
LIN {X -0.130,Y -554.230,Z 676.406,A 0.000,B 0.000,C 90.000,E1 289.014} C_DIS
LIN {X 0.110,Y -553.992,Z 676.399,A 0.000,B 0.000,C 90.000,E1 287.873} C_DIS
LIN {X 0.310,Y -553.408,Z 676.389,A 0.000,B 0.000,C 90.000,E1 285.898} C_DIS
LIN {X -0.032,Y -552.911,Z 676.381,A 0.000,B 0.000,C 90.000,E1 284.537} C_DIS
LIN {X 0.154,Y -552.210,Z 676.373,A 0.000,B 0.000,C 90.000,E1 283.119} C_DIS
LIN {X -0.218,Y -551.377,Z 676.364,A 0.000,B 0.000,C 90.000,E1 281.478} C_DIS
LIN {X 0.055,Y -550.326,Z 676.351,A 0.000,B 0.000,C 90.000,E1 279.208} C_DIS
LIN {X 0.207,Y -549.720,Z 676.339,A 0.000,B 0.000,C 90.000,E1 276.947} C_DIS
LIN {X 0.068,Y -549.443,Z 676.329,A 0.000,B 0.000,C 90.000,E1 275.277} C_DIS
LIN {X -0.123,Y -549.311,Z 676.320,A 0.000,B 0.000,C 90.000,E1 273.612} C_DIS
LIN {X 0.157,Y -549.085,Z 676.312,A 0.000,B 0.000,C 90.000,E1 272.178} C_DIS
LIN {X -0.170,Y -548.709,Z 676.306,A 0.000,B 0.000,C 90.000,E1 271.088} C_DIS
LIN {X 0.033,Y -548.183,Z 676.300,A 0.000,B 0.000,C 90.000,E1 269.943} C_DIS
LIN {X -0.228,Y -547.156,Z 676.290,A 0.000,B 0.000,C 90.000,E1 268.282} C_DIS
LIN {X 0.032,Y -546.374,Z 676.283,A 0.000,B 0.000,C 90.000,E1 266.846} C_DIS
LIN {X 0.250,Y -545.367,Z 676.275,A 0.000,B 0.000,C 90.000,E1 265.412} C_DIS
LIN {X 0.015,Y -544.045,Z 676.265,A 0.000,B 0.000,C 90.000,E1 263.742} C_DIS
LIN {X 0.201,Y -542.943,Z 676.259,A 0.000,B 0.000,C 90.000,E1 262.591} C_DIS
LIN {X 0.046,Y -540.821,Z 676.248,A 0.000,B 0.000,C 90.000,E1 260.622} C_DIS
LIN {X 0.032,Y -539.016,Z 676.237,A 0.000,B 0.000,C 90.000,E1 258.634} C_DIS
LIN {X 0.039,Y -537.078,Z 676.224,A 0.000,B 0.000,C 90.000,E1 256.353} C_DIS
LIN {X -0.119,Y -536.149,Z 676.218,A 0.000,B 0.000,C 90.000,E1 255.227} C_DIS
LIN {X -0.289,Y -535.023,Z 676.212,A 0.000,B 0.000,C 90.000,E1 254.102} C_DIS
LIN {X -0.097,Y -533.277,Z 676.202,A 0.000,B 0.000,C 90.000,E1 252.362} C_DIS
LIN {X -0.260,Y -531.304,Z 676.191,A 0.000,B 0.000,C 90.000,E1 250.369} C_DIS
LIN {X -0.179,Y -529.889,Z 676.184,A 0.000,B 0.000,C 90.000,E1 249.209} C_DIS
LIN {X 0.056,Y -527.873,Z 676.176,A 0.000,B 0.000,C 90.000,E1 247.741} C_DIS
LIN {X -0.037,Y -525.796,Z 676.168,A 0.000,B 0.000,C 90.000,E1 246.305} C_DIS
LIN {X 0.209,Y -522.847,Z 676.159,A 0.000,B 0.000,C 90.000,E1 244.537} C_DIS
LIN {X -0.047,Y -521.285,Z 676.154,A 0.000,B 0.000,C 90.000,E1 243.691} C_DIS
LIN {X -0.042,Y -518.389,Z 676.146,A 0.000,B 0.000,C 90.000,E1 242.231} C_DIS
LIN {X 0.026,Y -516.059,Z 676.139,A 0.000,B 0.000,C 90.000,E1 241.051} C_DIS
LIN {X 0.060,Y -513.550,Z 676.133,A 0.000,B 0.000,C 90.000,E1 239.871} C_DIS
LIN {X 0.313,Y -511.037,Z 676.126,A 0.000,B 0.000,C 90.000,E1 238.663} C_DIS
LIN {X 0.053,Y -507.100,Z 676.116,A 0.000,B 0.000,C 90.000,E1 236.914} C_DIS
LIN {X 0.260,Y -502.922,Z 676.106,A 0.000,B 0.000,C 90.000,E1 235.102} C_DIS
LIN {X -0.033,Y -498.506,Z 676.096,A 0.000,B 0.000,C 90.000,E1 233.336} C_DIS
LIN {X 0.012,Y -494.757,Z 676.088,A 0.000,B 0.000,C 90.000,E1 231.823} C_DIS
LIN {X 0.136,Y -490.401,Z 676.078,A 0.000,B 0.000,C 90.000,E1 229.989} C_DIS
LIN {X -0.049,Y -486.765,Z 676.069,A 0.000,B 0.000,C 90.000,E1 228.485} C_DIS
LIN {X 0.207,Y -483.856,Z 676.063,A 0.000,B 0.000,C 90.000,E1 227.229} C_DIS
LIN {X 0.120,Y -478.789,Z 676.051,A 0.000,B 0.000,C 90.000,E1 225.081} C_DIS
LIN {X 0.125,Y -474.390,Z 676.040,A 0.000,B 0.000,C 90.000,E1 223.218} C_DIS
LIN {X -0.041,Y -470.858,Z 676.032,A 0.000,B 0.000,C 90.000,E1 221.676} C_DIS
LIN {X -0.090,Y -466.158,Z 676.019,A 0.000,B 0.000,C 90.000,E1 219.483} C_DIS
LIN {X 0.046,Y -462.207,Z 676.009,A 0.000,B 0.000,C 90.000,E1 217.569} C_DIS
LIN {X -0.097,Y -458.388,Z 675.998,A 0.000,B 0.000,C 90.000,E1 215.678} C_DIS
LIN {X -0.060,Y -454.892,Z 675.988,A 0.000,B 0.000,C 90.000,E1 213.754} C_DIS
LIN {X 0.135,Y -451.181,Z 675.977,A 0.000,B 0.000,C 90.000,E1 211.799} C_DIS
LIN {X 0.093,Y -446.914,Z 675.964,A 0.000,B 0.000,C 90.000,E1 209.539} C_DIS
LIN {X 0.052,Y -443.379,Z 675.953,A 0.000,B 0.000,C 90.000,E1 207.590} C_DIS
LIN {X -0.112,Y -440.470,Z 675.944,A 0.000,B 0.000,C 90.000,E1 205.976} C_DIS
LIN {X -0.131,Y -437.448,Z 675.935,A 0.000,B 0.000,C 90.000,E1 204.335} C_DIS
LIN {X -0.043,Y -435.126,Z 675.928,A 0.000,B 0.000,C 90.000,E1 203.003} C_DIS
LIN {X -0.107,Y -432.109,Z 675.919,A 0.000,B 0.000,C 90.000,E1 201.354} C_DIS
LIN {X 0.138,Y -428.474,Z 675.907,A 0.000,B 0.000,C 90.000,E1 199.322} C_DIS
LIN {X 0.070,Y -424.377,Z 675.894,A 0.000,B 0.000,C 90.000,E1 196.985} C_DIS
LIN {X 0.061,Y -421.570,Z 675.885,A 0.000,B 0.000,C 90.000,E1 195.300} C_DIS
LIN {X 0.174,Y -418.659,Z 675.876,A 0.000,B 0.000,C 90.000,E1 193.592} C_DIS
LIN {X 0.015,Y -413.624,Z 675.859,A 0.000,B 0.000,C 90.000,E1 190.546} C_DIS
LIN {X -0.158,Y -410.420,Z 675.847,A 0.000,B 0.000,C 90.000,E1 188.511} C_DIS
LIN {X -0.066,Y -407.278,Z 675.836,A 0.000,B 0.000,C 90.000,E1 186.429} C_DIS
LIN {X 0.191,Y -403.109,Z 675.818,A 0.000,B 0.000,C 90.000,E1 183.269} C_DIS
LIN {X -0.051,Y -400.212,Z 675.805,A 0.000,B 0.000,C 90.000,E1 180.859} C_DIS
LIN {X 0.008,Y -397.882,Z 675.791,A 0.000,B 0.000,C 90.000,E1 178.396} C_DIS
LIN {X -0.131,Y -395.243,Z 675.772,A 0.000,B 0.000,C 90.000,E1 174.894} C_DIS
LIN {X -0.082,Y -394.003,Z 675.758,A 0.000,B 0.000,C 90.000,E1 172.413} C_DIS
LIN {X 0.006,Y -393.105,Z 675.742,A 0.000,B 0.000,C 90.000,E1 169.567} C_DIS
LIN {X -0.213,Y -392.710,Z 675.728,A 0.000,B 0.000,C 90.000,E1 167.117} C_DIS
LIN {X -0.134,Y -392.454,Z 675.713,A 0.000,B 0.000,C 90.000,E1 164.267} C_DIS
LIN {X -0.105,Y -392.458,Z 675.703,A 0.000,B 0.000,C 90.000,E1 162.489} C_DIS
LIN {X -0.170,Y -392.592,Z 675.691,A 0.000,B 0.000,C 90.000,E1 160.369} C_DIS
LIN {X 0.095,Y -392.872,Z 675.677,A 0.000,B 0.000,C 90.000,E1 157.847} C_DIS
LIN {X -0.050,Y -393.084,Z 675.665,A 0.000,B 0.000,C 90.000,E1 155.741} C_DIS
LIN {X -0.019,Y -393.511,Z 675.651,A 0.000,B 0.000,C 90.000,E1 153.256} C_DIS
LIN {X -0.148,Y -394.055,Z 675.638,A 0.000,B 0.000,C 90.000,E1 150.795} C_DIS
LIN {X 0.050,Y -394.482,Z 675.628,A 0.000,B 0.000,C 90.000,E1 148.997} C_DIS
LIN {X -0.212,Y -395.143,Z 675.616,A 0.000,B 0.000,C 90.000,E1 146.914} C_DIS
LIN {X 0.020,Y -396.665,Z 675.598,A 0.000,B 0.000,C 90.000,E1 143.703} C_DIS
LIN {X -0.068,Y -398.161,Z 675.585,A 0.000,B 0.000,C 90.000,E1 141.251} C_DIS
LIN {X 0.081,Y -399.923,Z 675.571,A 0.000,B 0.000,C 90.000,E1 138.771} C_DIS
LIN {X -0.070,Y -401.027,Z 675.563,A 0.000,B 0.000,C 90.000,E1 137.391} C_DIS
LIN {X -0.065,Y -403.310,Z 675.548,A 0.000,B 0.000,C 90.000,E1 134.595} C_DIS
LIN {X -0.011,Y -404.785,Z 675.542,A 0.000,B 0.000,C 90.000,E1 133.542} C_DIS
LIN {X 0.033,Y -405.983,Z 675.539,A 0.000,B 0.000,C 90.000,E1 133.014} C_DIS
LIN {X -0.207,Y -407.296,Z 675.537,A 0.000,B 0.000,C 90.000,E1 132.690} C_DIS
LIN {X -0.028,Y -408.323,Z 675.536,A 0.000,B 0.000,C 90.000,E1 132.405} C_DIS
LIN {X -0.069,Y -408.773,Z 675.535,A 0.000,B 0.000,C 90.000,E1 132.324} C_DIS
LIN {X -0.042,Y -411.626,Z 675.533,A 0.000,B 0.000,C 90.000,E1 131.881} C_DIS
LIN {X -0.147,Y -416.258,Z 675.530,A 0.000,B 0.000,C 90.000,E1 131.391} C_DIS
LIN {X 0.115,Y -436.559,Z 675.520,A 0.000,B 0.000,C 90.000,E1 129.644} C_DIS
LIN {X -0.248,Y -447.600,Z 675.516,A 0.000,B 0.000,C 90.000,E1 128.830} C_DIS
LIN {X -0.169,Y -463.362,Z 675.509,A 0.000,B 0.000,C 90.000,E1 127.604} C_DIS
LIN {X 0.185,Y -469.361,Z 675.506,A 0.000,B 0.000,C 90.000,E1 127.076} C_DIS
LIN {X -0.157,Y -478.214,Z 675.502,A 0.000,B 0.000,C 90.000,E1 126.377} C_DIS
LIN {X -0.063,Y -485.503,Z 675.498,A 0.000,B 0.000,C 90.000,E1 125.724} C_DIS
LIN {X 0.084,Y -489.861,Z 675.496,A 0.000,B 0.000,C 90.000,E1 125.311} C_DIS
LIN {X 0.080,Y -498.232,Z 675.492,A 0.000,B 0.000,C 90.000,E1 124.532} C_DIS
LIN {X 0.178,Y -507.670,Z 675.487,A 0.000,B 0.000,C 90.000,E1 123.579} C_DIS
LIN {X -0.007,Y -512.695,Z 675.484,A 0.000,B 0.000,C 90.000,E1 123.086} C_DIS
LIN {X -0.076,Y -517.737,Z 675.481,A 0.000,B 0.000,C 90.000,E1 122.546} C_DIS
LIN {X 0.026,Y -522.697,Z 675.478,A 0.000,B 0.000,C 90.000,E1 121.957} C_DIS
LIN {X -0.193,Y -526.415,Z 675.475,A 0.000,B 0.000,C 90.000,E1 121.544} C_DIS
LIN {X 0.174,Y -530.887,Z 675.472,A 0.000,B 0.000,C 90.000,E1 120.924} C_DIS
LIN {X -0.158,Y -535.003,Z 675.469,A 0.000,B 0.000,C 90.000,E1 120.384} C_DIS
LIN {X -0.141,Y -539.513,Z 675.465,A 0.000,B 0.000,C 90.000,E1 119.667} C_DIS
LIN {X -0.209,Y -544.281,Z 675.460,A 0.000,B 0.000,C 90.000,E1 118.821} C_DIS
LIN {X 0.023,Y -547.264,Z 675.457,A 0.000,B 0.000,C 90.000,E1 118.231} C_DIS
LIN {X 0.039,Y -551.218,Z 675.452,A 0.000,B 0.000,C 90.000,E1 117.385} C_DIS
LIN {X 0.094,Y -554.877,Z 675.448,A 0.000,B 0.000,C 90.000,E1 116.539} C_DIS
LIN {X 0.150,Y -557.193,Z 675.444,A 0.000,B 0.000,C 90.000,E1 115.976} C_DIS
LIN {X -0.188,Y -561.475,Z 675.438,A 0.000,B 0.000,C 90.000,E1 114.899} C_DIS
LIN {X -0.277,Y -564.387,Z 675.434,A 0.000,B 0.000,C 90.000,E1 114.079} C_DIS
LIN {X -0.006,Y -567.811,Z 675.428,A 0.000,B 0.000,C 90.000,E1 112.950} C_DIS
LIN {X 0.097,Y -570.698,Z 675.421,A 0.000,B 0.000,C 90.000,E1 111.844} C_DIS
LIN {X 0.269,Y -571.994,Z 675.418,A 0.000,B 0.000,C 90.000,E1 111.280} C_DIS
LIN {X 0.069,Y -573.765,Z 675.414,A 0.000,B 0.000,C 90.000,E1 110.482} C_DIS
LIN {X -0.115,Y -576.504,Z 675.406,A 0.000,B 0.000,C 90.000,E1 109.141} C_DIS
LIN {X 0.111,Y -579.133,Z 675.399,A 0.000,B 0.000,C 90.000,E1 107.764} C_DIS
LIN {X -0.161,Y -581.761,Z 675.391,A 0.000,B 0.000,C 90.000,E1 106.441} C_DIS
LIN {X -0.225,Y -583.848,Z 675.385,A 0.000,B 0.000,C 90.000,E1 105.371} C_DIS
LIN {X -0.018,Y -586.261,Z 675.378,A 0.000,B 0.000,C 90.000,E1 104.008} C_DIS
LIN {X 0.226,Y -588.624,Z 675.370,A 0.000,B 0.000,C 90.000,E1 102.647} C_DIS
LIN {X 0.109,Y -590.560,Z 675.365,A 0.000,B 0.000,C 90.000,E1 101.591} C_DIS
LIN {X 0.140,Y -593.860,Z 675.354,A 0.000,B 0.000,C 90.000,E1 99.726} C_DIS
LIN {X -0.135,Y -596.476,Z 675.345,A 0.000,B 0.000,C 90.000,E1 98.163} C_DIS
LIN {X -0.052,Y -598.455,Z 675.338,A 0.000,B 0.000,C 90.000,E1 96.834} C_DIS
LIN {X 0.000,Y -600.397,Z 675.331,A 0.000,B 0.000,C 90.000,E1 95.511} C_DIS
LIN {X 0.090,Y -602.128,Z 675.323,A 0.000,B 0.000,C 90.000,E1 94.188} C_DIS
LIN {X -0.081,Y -603.414,Z 675.318,A 0.000,B 0.000,C 90.000,E1 93.154} C_DIS
LIN {X 0.023,Y -604.762,Z 675.310,A 0.000,B 0.000,C 90.000,E1 91.835} C_DIS
LIN {X -0.122,Y -605.647,Z 675.304,A 0.000,B 0.000,C 90.000,E1 90.802} C_DIS
LIN {X -0.003,Y -606.501,Z 675.297,A 0.000,B 0.000,C 90.000,E1 89.484} C_DIS
LIN {X 0.196,Y -606.817,Z 675.293,A 0.000,B 0.000,C 90.000,E1 88.682} C_DIS
LIN {X -0.260,Y -607.230,Z 675.286,A 0.000,B 0.000,C 90.000,E1 87.421} C_DIS
LIN {X -0.104,Y -607.443,Z 675.278,A 0.000,B 0.000,C 90.000,E1 86.102} C_DIS
LIN {X 0.094,Y -607.372,Z 675.271,A 0.000,B 0.000,C 90.000,E1 84.780} C_DIS
LIN {X 0.036,Y -607.184,Z 675.265,A 0.000,B 0.000,C 90.000,E1 83.742} C_DIS
LIN {X 0.299,Y -606.714,Z 675.258,A 0.000,B 0.000,C 90.000,E1 82.413} C_DIS
LIN {X 0.225,Y -606.227,Z 675.252,A 0.000,B 0.000,C 90.000,E1 81.376} C_DIS
LIN {X 0.232,Y -605.361,Z 675.246,A 0.000,B 0.000,C 90.000,E1 80.330} C_DIS
LIN {X 0.271,Y -603.832,Z 675.238,A 0.000,B 0.000,C 90.000,E1 78.757} C_DIS
LIN {X -0.230,Y -602.673,Z 675.232,A 0.000,B 0.000,C 90.000,E1 77.757} C_DIS
LIN {X 0.156,Y -601.035,Z 675.225,A 0.000,B 0.000,C 90.000,E1 76.408} C_DIS
LIN {X 0.201,Y -599.642,Z 675.219,A 0.000,B 0.000,C 90.000,E1 75.353} C_DIS
LIN {X -0.203,Y -598.147,Z 675.213,A 0.000,B 0.000,C 90.000,E1 74.338} C_DIS
LIN {X -0.170,Y -596.140,Z 675.206,A 0.000,B 0.000,C 90.000,E1 73.015} C_DIS
LIN {X -0.164,Y -593.914,Z 675.198,A 0.000,B 0.000,C 90.000,E1 71.692} C_DIS
LIN {X 0.109,Y -592.052,Z 675.192,A 0.000,B 0.000,C 90.000,E1 70.604} C_DIS
LIN {X 0.230,Y -589.429,Z 675.185,A 0.000,B 0.000,C 90.000,E1 69.263} C_DIS
LIN {X -0.127,Y -587.040,Z 675.179,A 0.000,B 0.000,C 90.000,E1 68.230} C_DIS
LIN {X 0.048,Y -585.075,Z 675.175,A 0.000,B 0.000,C 90.000,E1 67.411} C_DIS
LIN {X -0.152,Y -582.113,Z 675.169,A 0.000,B 0.000,C 90.000,E1 66.357} C_DIS
LIN {X -0.158,Y -578.784,Z 675.163,A 0.000,B 0.000,C 90.000,E1 65.281} C_DIS
LIN {X -0.059,Y -576.128,Z 675.158,A 0.000,B 0.000,C 90.000,E1 64.460} C_DIS
LIN {X 0.008,Y -573.246,Z 675.154,A 0.000,B 0.000,C 90.000,E1 63.640} C_DIS
LIN {X 0.037,Y -570.204,Z 675.149,A 0.000,B 0.000,C 90.000,E1 62.820} C_DIS
LIN {X -0.210,Y -566.964,Z 675.145,A 0.000,B 0.000,C 90.000,E1 62.025} C_DIS
LIN {X -0.080,Y -562.741,Z 675.139,A 0.000,B 0.000,C 90.000,E1 61.051} C_DIS
LIN {X 0.292,Y -560.155,Z 675.136,A 0.000,B 0.000,C 90.000,E1 60.461} C_DIS
LIN {X 0.054,Y -556.471,Z 675.132,A 0.000,B 0.000,C 90.000,E1 59.793} C_DIS
LIN {X 0.145,Y -551.338,Z 675.128,A 0.000,B 0.000,C 90.000,E1 58.948} C_DIS
LIN {X -0.047,Y -547.632,Z 675.125,A 0.000,B 0.000,C 90.000,E1 58.408} C_DIS
LIN {X -0.134,Y -544.679,Z 675.122,A 0.000,B 0.000,C 90.000,E1 57.995} C_DIS
LIN {X 0.088,Y -540.302,Z 675.119,A 0.000,B 0.000,C 90.000,E1 57.406} C_DIS
LIN {X 0.270,Y -535.629,Z 675.116,A 0.000,B 0.000,C 90.000,E1 56.834} C_DIS
LIN {X 0.100,Y -529.291,Z 675.112,A 0.000,B 0.000,C 90.000,E1 56.215} C_DIS
LIN {X 0.235,Y -524.869,Z 675.110,A 0.000,B 0.000,C 90.000,E1 55.801} C_DIS
LIN {X 0.065,Y -518.680,Z 675.108,A 0.000,B 0.000,C 90.000,E1 55.341} C_DIS
LIN {X -0.135,Y -513.964,Z 675.106,A 0.000,B 0.000,C 90.000,E1 55.022} C_DIS
LIN {X -0.066,Y -509.061,Z 675.104,A 0.000,B 0.000,C 90.000,E1 54.689} C_DIS
LIN {X -0.162,Y -500.751,Z 675.101,A 0.000,B 0.000,C 90.000,E1 54.196} C_DIS
LIN {X 0.099,Y -493.939,Z 675.099,A 0.000,B 0.000,C 90.000,E1 53.783} C_DIS
LIN {X 0.032,Y -475.970,Z 675.093,A 0.000,B 0.000,C 90.000,E1 52.798} C_DIS
LIN {X 0.005,Y -462.767,Z 675.089,A 0.000,B 0.000,C 90.000,E1 52.065} C_DIS
LIN {X -0.057,Y -443.122,Z 675.083,A 0.000,B 0.000,C 90.000,E1 50.928} C_DIS
LIN {X -0.098,Y -429.603,Z 675.078,A 0.000,B 0.000,C 90.000,E1 50.070} C_DIS
LIN {X -0.122,Y -429.584,Z 675.078,A 0.000,B 0.000,C 90.000,E1 50.070} C_DIS
LIN {X -0.086,Y -420.676,Z 675.055,A 0.000,B 0.000,C 90.000,E1 45.972} C_DIS
LIN {X 0.184,Y -418.856,Z 675.050,A 0.000,B 0.000,C 90.000,E1 44.919} C_DIS
LIN {X -0.159,Y -416.481,Z 675.044,A 0.000,B 0.000,C 90.000,E1 43.947} C_DIS
LIN {X -0.009,Y -415.551,Z 675.042,A 0.000,B 0.000,C 90.000,E1 43.500} C_DIS
LIN {X -0.030,Y -415.584,Z 675.033,A 0.000,B 0.000,C 90.000,E1 41.881} C_DIS
LIN {X 0.157,Y -415.796,Z 675.021,A 0.000,B 0.000,C 90.000,E1 39.806} C_DIS
LIN {X -0.127,Y -417.069,Z 675.000,A 0.000,B 0.000,C 90.000,E1 36.091} C_DIS
LIN {X 0.136,Y -417.784,Z 674.993,A 0.000,B 0.000,C 90.000,E1 34.692} C_DIS
LIN {X -0.121,Y -419.188,Z 674.978,A 0.000,B 0.000,C 90.000,E1 32.005} C_DIS
LIN {X -0.280,Y -419.953,Z 674.970,A 0.000,B 0.000,C 90.000,E1 30.669} C_DIS
LIN {X -0.138,Y -421.048,Z 674.959,A 0.000,B 0.000,C 90.000,E1 28.615} C_DIS
LIN {X 0.231,Y -422.081,Z 674.950,A 0.000,B 0.000,C 90.000,E1 26.873} C_DIS
LIN {X 0.052,Y -423.211,Z 674.940,A 0.000,B 0.000,C 90.000,E1 25.207} C_DIS
LIN {X 0.008,Y -426.146,Z 674.921,A 0.000,B 0.000,C 90.000,E1 21.844} C_DIS
LIN {X -0.055,Y -427.757,Z 674.912,A 0.000,B 0.000,C 90.000,E1 20.174} C_DIS
LIN {X 0.151,Y -428.606,Z 674.906,A 0.000,B 0.000,C 90.000,E1 19.141} C_DIS
LIN {X -0.162,Y -429.968,Z 674.897,A 0.000,B 0.000,C 90.000,E1 17.511} C_DIS
LIN {X -0.050,Y -432.132,Z 674.882,A 0.000,B 0.000,C 90.000,E1 14.828} C_DIS
LIN {X 0.120,Y -434.427,Z 674.869,A 0.000,B 0.000,C 90.000,E1 12.479} C_DIS
LIN {X -0.129,Y -435.860,Z 674.862,A 0.000,B 0.000,C 90.000,E1 11.186} C_DIS
LIN {X 0.123,Y -438.765,Z 674.847,A 0.000,B 0.000,C 90.000,E1 8.511} C_DIS
LIN {X 0.185,Y -441.591,Z 674.835,A 0.000,B 0.000,C 90.000,E1 6.201} C_DIS
LIN {X -0.042,Y -445.055,Z 674.820,A 0.000,B 0.000,C 90.000,E1 3.612} C_DIS
LIN {X -0.226,Y -447.452,Z 674.811,A 0.000,B 0.000,C 90.000,E1 2.007} C_DIS
LIN {X 0.042,Y -451.922,Z 674.795,A 0.000,B 0.000,C 90.000,E1 359.141} C_DIS
LIN {X 0.164,Y -455.377,Z 674.785,A 0.000,B 0.000,C 90.000,E1 357.192} C_DIS
LIN {X 0.205,Y -458.325,Z 674.776,A 0.000,B 0.000,C 90.000,E1 355.584} C_DIS
LIN {X -0.160,Y -461.329,Z 674.767,A 0.000,B 0.000,C 90.000,E1 354.033} C_DIS
LIN {X -0.178,Y -464.874,Z 674.756,A 0.000,B 0.000,C 90.000,E1 352.129} C_DIS
LIN {X 0.217,Y -467.829,Z 674.747,A 0.000,B 0.000,C 90.000,E1 350.500} C_DIS
LIN {X -0.150,Y -470.104,Z 674.740,A 0.000,B 0.000,C 90.000,E1 349.285} C_DIS
LIN {X -0.020,Y -472.892,Z 674.732,A 0.000,B 0.000,C 90.000,E1 347.701} C_DIS
LIN {X 0.002,Y -476.270,Z 674.721,A 0.000,B 0.000,C 90.000,E1 345.825} C_DIS
LIN {X -0.281,Y -480.346,Z 674.709,A 0.000,B 0.000,C 90.000,E1 343.685} C_DIS
LIN {X -0.173,Y -483.914,Z 674.699,A 0.000,B 0.000,C 90.000,E1 341.819} C_DIS
LIN {X 0.031,Y -488.273,Z 674.687,A 0.000,B 0.000,C 90.000,E1 339.645} C_DIS
LIN {X 0.162,Y -491.386,Z 674.679,A 0.000,B 0.000,C 90.000,E1 338.103} C_DIS
LIN {X -0.104,Y -494.331,Z 674.670,A 0.000,B 0.000,C 90.000,E1 336.613} C_DIS
LIN {X -0.116,Y -497.160,Z 674.662,A 0.000,B 0.000,C 90.000,E1 335.101} C_DIS
LIN {X -0.078,Y -500.203,Z 674.653,A 0.000,B 0.000,C 90.000,E1 333.589} C_DIS
LIN {X -0.184,Y -501.818,Z 674.650,A 0.000,B 0.000,C 90.000,E1 332.999} C_DIS
LIN {X 0.171,Y -503.853,Z 674.647,A 0.000,B 0.000,C 90.000,E1 332.359} C_DIS
LIN {X 0.268,Y -504.772,Z 674.646,A 0.000,B 0.000,C 90.000,E1 332.153} C_DIS
LIN {X 0.151,Y -507.700,Z 674.643,A 0.000,B 0.000,C 90.000,E1 331.719} C_DIS
LIN {X -0.059,Y -511.653,Z 674.641,A 0.000,B 0.000,C 90.000,E1 331.307} C_DIS
LIN {X 0.028,Y -515.019,Z 674.639,A 0.000,B 0.000,C 90.000,E1 331.001} C_DIS
LIN {X -0.151,Y -533.159,Z 674.632,A 0.000,B 0.000,C 90.000,E1 329.744} C_DIS
LIN {X -0.013,Y -537.581,Z 674.630,A 0.000,B 0.000,C 90.000,E1 329.410} C_DIS
LIN {X -0.213,Y -546.394,Z 674.626,A 0.000,B 0.000,C 90.000,E1 328.742} C_DIS
LIN {X 0.128,Y -553.307,Z 674.623,A 0.000,B 0.000,C 90.000,E1 328.122} C_DIS
LIN {X 0.150,Y -562.836,Z 674.618,A 0.000,B 0.000,C 90.000,E1 327.248} C_DIS
LIN {X -0.101,Y -572.033,Z 674.613,A 0.000,B 0.000,C 90.000,E1 326.373} C_DIS
LIN {X -0.166,Y -581.048,Z 674.608,A 0.000,B 0.000,C 90.000,E1 325.468} C_DIS
LIN {X -0.152,Y -589.918,Z 674.603,A 0.000,B 0.000,C 90.000,E1 324.562} C_DIS
LIN {X -0.160,Y -596.063,Z 674.599,A 0.000,B 0.000,C 90.000,E1 323.909} C_DIS
LIN {X -0.268,Y -603.204,Z 674.595,A 0.000,B 0.000,C 90.000,E1 323.130} C_DIS
LIN {X 0.034,Y -609.944,Z 674.591,A 0.000,B 0.000,C 90.000,E1 322.316} C_DIS
LIN {X 0.271,Y -613.127,Z 674.589,A 0.000,B 0.000,C 90.000,E1 321.904} C_DIS
LIN {X 0.130,Y -620.883,Z 674.583,A 0.000,B 0.000,C 90.000,E1 320.884} C_DIS
LIN {X 0.295,Y -624.502,Z 674.580,A 0.000,B 0.000,C 90.000,E1 320.356} C_DIS
LIN {X 0.038,Y -628.805,Z 674.576,A 0.000,B 0.000,C 90.000,E1 319.747} C_DIS
LIN {X 0.234,Y -632.960,Z 674.573,A 0.000,B 0.000,C 90.000,E1 319.094} C_DIS
LIN {X -0.096,Y -637.690,Z 674.569,A 0.000,B 0.000,C 90.000,E1 318.366} C_DIS
LIN {X -0.413,Y -643.717,Z 674.563,A 0.000,B 0.000,C 90.000,E1 317.391} C_DIS
LIN {X -0.226,Y -649.351,Z 674.558,A 0.000,B 0.000,C 90.000,E1 316.377} C_DIS
LIN {X 0.052,Y -654.087,Z 674.553,A 0.000,B 0.000,C 90.000,E1 315.486} C_DIS
LIN {X -0.090,Y -659.074,Z 674.547,A 0.000,B 0.000,C 90.000,E1 314.514} C_DIS
LIN {X -0.192,Y -664.896,Z 674.541,A 0.000,B 0.000,C 90.000,E1 313.299} C_DIS
LIN {X -0.172,Y -670.395,Z 674.534,A 0.000,B 0.000,C 90.000,E1 312.081} C_DIS
LIN {X -0.148,Y -673.574,Z 674.530,A 0.000,B 0.000,C 90.000,E1 311.353} C_DIS
LIN {X -0.013,Y -677.566,Z 674.524,A 0.000,B 0.000,C 90.000,E1 310.378} C_DIS
LIN {X 0.147,Y -680.277,Z 674.520,A 0.000,B 0.000,C 90.000,E1 309.644} C_DIS
LIN {X 0.339,Y -682.715,Z 674.516,A 0.000,B 0.000,C 90.000,E1 308.910} C_DIS
LIN {X 0.172,Y -685.699,Z 674.511,A 0.000,B 0.000,C 90.000,E1 307.971} C_DIS
LIN {X 0.044,Y -688.350,Z 674.506,A 0.000,B 0.000,C 90.000,E1 307.030} C_DIS
LIN {X -0.055,Y -690.772,Z 674.501,A 0.000,B 0.000,C 90.000,E1 306.091} C_DIS
LIN {X -0.133,Y -692.941,Z 674.495,A 0.000,B 0.000,C 90.000,E1 305.152} C_DIS
LIN {X -0.016,Y -694.879,Z 674.490,A 0.000,B 0.000,C 90.000,E1 304.199} C_DIS
LIN {X 0.136,Y -696.626,Z 674.485,A 0.000,B 0.000,C 90.000,E1 303.245} C_DIS
LIN {X 0.067,Y -697.776,Z 674.481,A 0.000,B 0.000,C 90.000,E1 302.546} C_DIS
LIN {X -0.089,Y -699.427,Z 674.474,A 0.000,B 0.000,C 90.000,E1 301.386} C_DIS
LIN {X -0.249,Y -700.575,Z 674.469,A 0.000,B 0.000,C 90.000,E1 300.463} C_DIS
LIN {X -0.390,Y -701.486,Z 674.464,A 0.000,B 0.000,C 90.000,E1 299.539} C_DIS
LIN {X 0.095,Y -702.288,Z 674.459,A 0.000,B 0.000,C 90.000,E1 298.565} C_DIS
LIN {X -0.129,Y -703.575,Z 674.450,A 0.000,B 0.000,C 90.000,E1 296.950} C_DIS
LIN {X 0.032,Y -704.391,Z 674.443,A 0.000,B 0.000,C 90.000,E1 295.771} C_DIS
LIN {X 0.013,Y -704.408,Z 674.442,A 0.000,B 0.000,C 90.000,E1 295.540} C_DIS
LIN {X -0.051,Y -703.999,Z 674.439,A 0.000,B 0.000,C 90.000,E1 295.079} C_DIS
LIN {X -0.063,Y -703.427,Z 674.438,A 0.000,B 0.000,C 90.000,E1 294.847} C_DIS
LIN {X -0.136,Y -701.462,Z 674.435,A 0.000,B 0.000,C 90.000,E1 294.387} C_DIS
LIN {X 0.002,Y -700.815,Z 674.435,A 0.000,B 0.000,C 90.000,E1 294.259} C_DIS
LIN {X 0.140,Y -699.841,Z 674.434,A 0.000,B 0.000,C 90.000,E1 294.131} C_DIS
LIN {X 0.125,Y -696.830,Z 674.433,A 0.000,B 0.000,C 90.000,E1 293.898} C_DIS
LIN {X 0.148,Y -694.001,Z 674.432,A 0.000,B 0.000,C 90.000,E1 293.695} C_DIS
LIN {X 0.235,Y -692.437,Z 674.431,A 0.000,B 0.000,C 90.000,E1 293.590} C_DIS
LIN {X -0.036,Y -689.917,Z 674.431,A 0.000,B 0.000,C 90.000,E1 293.515} C_DIS
LIN {X -0.183,Y -687.741,Z 674.430,A 0.000,B 0.000,C 90.000,E1 293.462} C_DIS
LIN {X 0.056,Y -679.965,Z 674.429,A 0.000,B 0.000,C 90.000,E1 293.259} C_DIS
LIN {X 0.092,Y -664.544,Z 674.428,A 0.000,B 0.000,C 90.000,E1 293.078} C_DIS
LIN {X -0.013,Y -651.379,Z 674.427,A 0.000,B 0.000,C 90.000,E1 292.898} C_DIS
LIN {X 0.101,Y -638.161,Z 674.426,A 0.000,B 0.000,C 90.000,E1 292.642} C_DIS
LIN {X -0.324,Y -628.207,Z 674.425,A 0.000,B 0.000,C 90.000,E1 292.461} C_DIS
LIN {X 0.103,Y -614.825,Z 674.423,A 0.000,B 0.000,C 90.000,E1 292.078} C_DIS
LIN {X 0.181,Y -594.340,Z 674.419,A 0.000,B 0.000,C 90.000,E1 291.461} C_DIS
LIN {X 0.102,Y -576.952,Z 674.416,A 0.000,B 0.000,C 90.000,E1 290.918} C_DIS
LIN {X -0.164,Y -562.751,Z 674.414,A 0.000,B 0.000,C 90.000,E1 290.536} C_DIS
LIN {X -0.182,Y -556.775,Z 674.412,A 0.000,B 0.000,C 90.000,E1 290.248} C_DIS
LIN {X -0.231,Y -556.707,Z 674.412,A 0.000,B 0.000,C 90.000,E1 290.248} C_DIS
LIN {X 0.000,Y -555.371,Z 674.411,A 0.000,B 0.000,C 90.000,E1 290.066} C_DIS
LIN {X -0.042,Y -555.343,Z 674.411,A 0.000,B 0.000,C 90.000,E1 290.066} C_DIS
LIN {X -0.056,Y -554.869,Z 674.410,A 0.000,B 0.000,C 90.000,E1 289.885} C_DIS
LIN {X -0.072,Y -554.520,Z 674.409,A 0.000,B 0.000,C 90.000,E1 289.631} C_DIS
LIN {X -0.146,Y -554.237,Z 674.405,A 0.000,B 0.000,C 90.000,E1 288.833} C_DIS
LIN {X 0.203,Y -553.888,Z 674.397,A 0.000,B 0.000,C 90.000,E1 287.402} C_DIS
LIN {X 0.026,Y -553.470,Z 674.389,A 0.000,B 0.000,C 90.000,E1 286.024} C_DIS
LIN {X -0.169,Y -552.978,Z 674.381,A 0.000,B 0.000,C 90.000,E1 284.647} C_DIS
LIN {X -0.114,Y -552.329,Z 674.374,A 0.000,B 0.000,C 90.000,E1 283.244} C_DIS
LIN {X 0.176,Y -551.451,Z 674.364,A 0.000,B 0.000,C 90.000,E1 281.535} C_DIS
LIN {X -0.096,Y -550.408,Z 674.352,A 0.000,B 0.000,C 90.000,E1 279.321} C_DIS
LIN {X -0.015,Y -549.779,Z 674.339,A 0.000,B 0.000,C 90.000,E1 277.068} C_DIS
LIN {X -0.184,Y -549.540,Z 674.331,A 0.000,B 0.000,C 90.000,E1 275.682} C_DIS
LIN {X 0.267,Y -549.359,Z 674.321,A 0.000,B 0.000,C 90.000,E1 273.669} C_DIS
LIN {X -0.003,Y -549.139,Z 674.313,A 0.000,B 0.000,C 90.000,E1 272.293} C_DIS
LIN {X 0.169,Y -548.892,Z 674.308,A 0.000,B 0.000,C 90.000,E1 271.432} C_DIS
LIN {X -0.124,Y -548.259,Z 674.300,A 0.000,B 0.000,C 90.000,E1 270.057} C_DIS
LIN {X 0.164,Y -547.279,Z 674.291,A 0.000,B 0.000,C 90.000,E1 268.339} C_DIS
LIN {X -0.079,Y -546.312,Z 674.282,A 0.000,B 0.000,C 90.000,E1 266.674} C_DIS
LIN {X 0.209,Y -545.066,Z 674.272,A 0.000,B 0.000,C 90.000,E1 264.951} C_DIS
LIN {X -0.107,Y -543.916,Z 674.264,A 0.000,B 0.000,C 90.000,E1 263.571} C_DIS
LIN {X 0.144,Y -542.800,Z 674.258,A 0.000,B 0.000,C 90.000,E1 262.413} C_DIS
LIN {X -0.081,Y -540.958,Z 674.249,A 0.000,B 0.000,C 90.000,E1 260.735} C_DIS
LIN {X -0.121,Y -538.863,Z 674.236,A 0.000,B 0.000,C 90.000,E1 258.465} C_DIS
LIN {X -0.064,Y -537.198,Z 674.225,A 0.000,B 0.000,C 90.000,E1 256.464} C_DIS
LIN {X 0.303,Y -536.274,Z 674.218,A 0.000,B 0.000,C 90.000,E1 255.283} C_DIS
LIN {X 0.183,Y -534.912,Z 674.211,A 0.000,B 0.000,C 90.000,E1 253.866} C_DIS
LIN {X 0.055,Y -532.829,Z 674.199,A 0.000,B 0.000,C 90.000,E1 251.873} C_DIS
LIN {X 0.181,Y -531.453,Z 674.191,A 0.000,B 0.000,C 90.000,E1 250.423} C_DIS
LIN {X 0.266,Y -530.078,Z 674.185,A 0.000,B 0.000,C 90.000,E1 249.263} C_DIS
LIN {X 0.019,Y -528.054,Z 674.177,A 0.000,B 0.000,C 90.000,E1 247.847} C_DIS
LIN {X -0.061,Y -526.007,Z 674.169,A 0.000,B 0.000,C 90.000,E1 246.410} C_DIS
LIN {X -0.021,Y -523.054,Z 674.159,A 0.000,B 0.000,C 90.000,E1 244.665} C_DIS
LIN {X -0.127,Y -520.931,Z 674.153,A 0.000,B 0.000,C 90.000,E1 243.512} C_DIS
LIN {X -0.224,Y -517.468,Z 674.143,A 0.000,B 0.000,C 90.000,E1 241.769} C_DIS
LIN {X -0.167,Y -515.067,Z 674.137,A 0.000,B 0.000,C 90.000,E1 240.589} C_DIS
LIN {X 0.108,Y -511.236,Z 674.127,A 0.000,B 0.000,C 90.000,E1 238.791} C_DIS
LIN {X -0.043,Y -507.975,Z 674.119,A 0.000,B 0.000,C 90.000,E1 237.327} C_DIS
LIN {X 0.291,Y -504.547,Z 674.110,A 0.000,B 0.000,C 90.000,E1 235.801} C_DIS
LIN {X -0.026,Y -501.662,Z 674.104,A 0.000,B 0.000,C 90.000,E1 234.642} C_DIS
LIN {X -0.057,Y -497.193,Z 674.094,A 0.000,B 0.000,C 90.000,E1 232.844} C_DIS
LIN {X -0.024,Y -492.039,Z 674.082,A 0.000,B 0.000,C 90.000,E1 230.723} C_DIS
LIN {X -0.173,Y -488.410,Z 674.073,A 0.000,B 0.000,C 90.000,E1 229.218} C_DIS
LIN {X -0.211,Y -485.479,Z 674.067,A 0.000,B 0.000,C 90.000,E1 228.000} C_DIS
LIN {X -0.165,Y -481.830,Z 674.058,A 0.000,B 0.000,C 90.000,E1 226.458} C_DIS
LIN {X 0.012,Y -478.965,Z 674.051,A 0.000,B 0.000,C 90.000,E1 225.202} C_DIS
LIN {X 0.253,Y -475.279,Z 674.043,A 0.000,B 0.000,C 90.000,E1 223.623} C_DIS
LIN {X 0.195,Y -471.026,Z 674.032,A 0.000,B 0.000,C 90.000,E1 221.757} C_DIS
LIN {X 0.150,Y -466.317,Z 674.020,A 0.000,B 0.000,C 90.000,E1 219.564} C_DIS
LIN {X 0.007,Y -462.390,Z 674.009,A 0.000,B 0.000,C 90.000,E1 217.684} C_DIS
LIN {X 0.157,Y -457.921,Z 673.997,A 0.000,B 0.000,C 90.000,E1 215.438} C_DIS
LIN {X -0.060,Y -454.993,Z 673.988,A 0.000,B 0.000,C 90.000,E1 213.865} C_DIS
LIN {X 0.011,Y -451.309,Z 673.977,A 0.000,B 0.000,C 90.000,E1 211.926} C_DIS
LIN {X -0.030,Y -447.044,Z 673.965,A 0.000,B 0.000,C 90.000,E1 209.667} C_DIS
LIN {X -0.014,Y -442.963,Z 673.952,A 0.000,B 0.000,C 90.000,E1 207.385} C_DIS
LIN {X 0.047,Y -439.410,Z 673.941,A 0.000,B 0.000,C 90.000,E1 205.412} C_DIS
LIN {X -0.156,Y -435.917,Z 673.930,A 0.000,B 0.000,C 90.000,E1 203.462} C_DIS
LIN {X -0.053,Y -432.257,Z 673.919,A 0.000,B 0.000,C 90.000,E1 201.461} C_DIS
LIN {X 0.044,Y -428.649,Z 673.908,A 0.000,B 0.000,C 90.000,E1 199.450} C_DIS
LIN {X -0.228,Y -423.991,Z 673.893,A 0.000,B 0.000,C 90.000,E1 196.804} C_DIS
LIN {X 0.162,Y -421.156,Z 673.884,A 0.000,B 0.000,C 90.000,E1 195.064} C_DIS
LIN {X -0.139,Y -418.259,Z 673.874,A 0.000,B 0.000,C 90.000,E1 193.411} C_DIS
LIN {X 0.046,Y -413.802,Z 673.859,A 0.000,B 0.000,C 90.000,E1 190.658} C_DIS
LIN {X -0.161,Y -411.166,Z 673.850,A 0.000,B 0.000,C 90.000,E1 188.973} C_DIS
LIN {X -0.052,Y -408.004,Z 673.838,A 0.000,B 0.000,C 90.000,E1 186.891} C_DIS
LIN {X -0.138,Y -404.164,Z 673.823,A 0.000,B 0.000,C 90.000,E1 184.131} C_DIS
LIN {X 0.099,Y -401.613,Z 673.811,A 0.000,B 0.000,C 90.000,E1 182.007} C_DIS
LIN {X 0.052,Y -398.061,Z 673.792,A 0.000,B 0.000,C 90.000,E1 178.511} C_DIS
LIN {X -0.077,Y -395.414,Z 673.772,A 0.000,B 0.000,C 90.000,E1 175.008} C_DIS
LIN {X -0.112,Y -394.006,Z 673.757,A 0.000,B 0.000,C 90.000,E1 172.186} C_DIS
LIN {X 0.047,Y -393.317,Z 673.745,A 0.000,B 0.000,C 90.000,E1 170.038} C_DIS
LIN {X -0.170,Y -392.853,Z 673.731,A 0.000,B 0.000,C 90.000,E1 167.589} C_DIS
LIN {X -0.135,Y -392.687,Z 673.721,A 0.000,B 0.000,C 90.000,E1 165.811} C_DIS
LIN {X -0.101,Y -392.657,Z 673.707,A 0.000,B 0.000,C 90.000,E1 163.323} C_DIS
LIN {X -0.232,Y -392.768,Z 673.694,A 0.000,B 0.000,C 90.000,E1 160.859} C_DIS
LIN {X 0.159,Y -392.914,Z 673.684,A 0.000,B 0.000,C 90.000,E1 159.028} C_DIS
LIN {X -0.030,Y -393.144,Z 673.674,A 0.000,B 0.000,C 90.000,E1 157.283} C_DIS
LIN {X 0.035,Y -393.474,Z 673.660,A 0.000,B 0.000,C 90.000,E1 154.793} C_DIS
LIN {X 0.046,Y -393.858,Z 673.648,A 0.000,B 0.000,C 90.000,E1 152.666} C_DIS
LIN {X -0.140,Y -394.302,Z 673.638,A 0.000,B 0.000,C 90.000,E1 150.923} C_DIS
LIN {X -0.068,Y -394.761,Z 673.627,A 0.000,B 0.000,C 90.000,E1 148.791} C_DIS
LIN {X -0.191,Y -395.398,Z 673.617,A 0.000,B 0.000,C 90.000,E1 147.041} C_DIS
LIN {X 0.056,Y -396.836,Z 673.599,A 0.000,B 0.000,C 90.000,E1 143.829} C_DIS
LIN {X -0.020,Y -398.255,Z 673.585,A 0.000,B 0.000,C 90.000,E1 141.376} C_DIS
LIN {X 0.070,Y -399.678,Z 673.574,A 0.000,B 0.000,C 90.000,E1 139.256} C_DIS
LIN {X -0.005,Y -401.034,Z 673.564,A 0.000,B 0.000,C 90.000,E1 137.514} C_DIS
LIN {X 0.123,Y -403.533,Z 673.547,A 0.000,B 0.000,C 90.000,E1 134.352} C_DIS
LIN {X -0.222,Y -404.473,Z 673.543,A 0.000,B 0.000,C 90.000,E1 133.704} C_DIS
LIN {X 0.224,Y -406.110,Z 673.538,A 0.000,B 0.000,C 90.000,E1 132.771} C_DIS
LIN {X -0.006,Y -408.271,Z 673.535,A 0.000,B 0.000,C 90.000,E1 132.243} C_DIS
LIN {X -0.087,Y -409.060,Z 673.534,A 0.000,B 0.000,C 90.000,E1 132.081} C_DIS
LIN {X -0.249,Y -411.266,Z 673.532,A 0.000,B 0.000,C 90.000,E1 131.757} C_DIS
LIN {X -0.023,Y -415.789,Z 673.529,A 0.000,B 0.000,C 90.000,E1 131.229} C_DIS
LIN {X 0.092,Y -421.542,Z 673.526,A 0.000,B 0.000,C 90.000,E1 130.701} C_DIS
LIN {X -0.075,Y -427.605,Z 673.523,A 0.000,B 0.000,C 90.000,E1 130.216} C_DIS
LIN {X -0.002,Y -443.322,Z 673.516,A 0.000,B 0.000,C 90.000,E1 128.955} C_DIS
LIN {X 0.097,Y -455.969,Z 673.511,A 0.000,B 0.000,C 90.000,E1 127.971} C_DIS
LIN {X 0.204,Y -463.779,Z 673.508,A 0.000,B 0.000,C 90.000,E1 127.363} C_DIS
LIN {X 0.254,Y -469.860,Z 673.505,A 0.000,B 0.000,C 90.000,E1 126.870} C_DIS
LIN {X -0.207,Y -477.413,Z 673.502,A 0.000,B 0.000,C 90.000,E1 126.297} C_DIS
LIN {X -0.069,Y -484.762,Z 673.498,A 0.000,B 0.000,C 90.000,E1 125.644} C_DIS
LIN {X 0.072,Y -490.554,Z 673.495,A 0.000,B 0.000,C 90.000,E1 125.105} C_DIS
LIN {X -0.025,Y -497.748,Z 673.491,A 0.000,B 0.000,C 90.000,E1 124.452} C_DIS
LIN {X -0.102,Y -508.703,Z 673.485,A 0.000,B 0.000,C 90.000,E1 123.372} C_DIS
LIN {X -0.031,Y -512.718,Z 673.483,A 0.000,B 0.000,C 90.000,E1 122.959} C_DIS
LIN {X -0.186,Y -517.877,Z 673.480,A 0.000,B 0.000,C 90.000,E1 122.418} C_DIS
LIN {X 0.069,Y -524.132,Z 673.476,A 0.000,B 0.000,C 90.000,E1 121.671} C_DIS
LIN {X -0.146,Y -527.717,Z 673.474,A 0.000,B 0.000,C 90.000,E1 121.258} C_DIS
LIN {X 0.109,Y -531.117,Z 673.471,A 0.000,B 0.000,C 90.000,E1 120.797} C_DIS
LIN {X -0.222,Y -535.259,Z 673.468,A 0.000,B 0.000,C 90.000,E1 120.256} C_DIS
LIN {X -0.061,Y -538.980,Z 673.465,A 0.000,B 0.000,C 90.000,E1 119.667} C_DIS
LIN {X 0.018,Y -543.796,Z 673.460,A 0.000,B 0.000,C 90.000,E1 118.821} C_DIS
LIN {X 0.244,Y -546.875,Z 673.457,A 0.000,B 0.000,C 90.000,E1 118.231} C_DIS
LIN {X 0.258,Y -550.931,Z 673.452,A 0.000,B 0.000,C 90.000,E1 117.385} C_DIS
LIN {X -0.046,Y -555.252,Z 673.447,A 0.000,B 0.000,C 90.000,E1 116.437} C_DIS
LIN {X 0.155,Y -558.114,Z 673.443,A 0.000,B 0.000,C 90.000,E1 115.720} C_DIS
LIN {X 0.032,Y -561.368,Z 673.438,A 0.000,B 0.000,C 90.000,E1 114.899} C_DIS
LIN {X -0.056,Y -564.329,Z 673.434,A 0.000,B 0.000,C 90.000,E1 114.079} C_DIS
LIN {X 0.215,Y -567.796,Z 673.428,A 0.000,B 0.000,C 90.000,E1 112.950} C_DIS
LIN {X -0.029,Y -570.066,Z 673.423,A 0.000,B 0.000,C 90.000,E1 112.153} C_DIS
LIN {X 0.139,Y -571.482,Z 673.420,A 0.000,B 0.000,C 90.000,E1 111.589} C_DIS
LIN {X -0.067,Y -573.365,Z 673.416,A 0.000,B 0.000,C 90.000,E1 110.791} C_DIS
LIN {X -0.256,Y -576.174,Z 673.408,A 0.000,B 0.000,C 90.000,E1 109.450} C_DIS
LIN {X -0.207,Y -579.354,Z 673.399,A 0.000,B 0.000,C 90.000,E1 107.819} C_DIS
LIN {X -0.261,Y -582.562,Z 673.390,A 0.000,B 0.000,C 90.000,E1 106.205} C_DIS
LIN {X -0.313,Y -584.635,Z 673.384,A 0.000,B 0.000,C 90.000,E1 105.134} C_DIS
LIN {X 0.159,Y -587.566,Z 673.375,A 0.000,B 0.000,C 90.000,E1 103.480} C_DIS
LIN {X 0.109,Y -590.486,Z 673.366,A 0.000,B 0.000,C 90.000,E1 101.883} C_DIS
LIN {X -0.171,Y -594.289,Z 673.354,A 0.000,B 0.000,C 90.000,E1 99.782} C_DIS
LIN {X 0.150,Y -596.957,Z 673.345,A 0.000,B 0.000,C 90.000,E1 98.163} C_DIS
LIN {X 0.241,Y -598.968,Z 673.338,A 0.000,B 0.000,C 90.000,E1 96.834} C_DIS
LIN {X -0.005,Y -601.308,Z 673.329,A 0.000,B 0.000,C 90.000,E1 95.277} C_DIS
LIN {X 0.092,Y -603.031,Z 673.322,A 0.000,B 0.000,C 90.000,E1 93.955} C_DIS
LIN {X -0.076,Y -604.290,Z 673.316,A 0.000,B 0.000,C 90.000,E1 92.922} C_DIS
LIN {X 0.032,Y -605.600,Z 673.309,A 0.000,B 0.000,C 90.000,E1 91.604} C_DIS
LIN {X -0.119,Y -606.435,Z 673.303,A 0.000,B 0.000,C 90.000,E1 90.573} C_DIS
LIN {X -0.256,Y -607.142,Z 673.297,A 0.000,B 0.000,C 90.000,E1 89.542} C_DIS
LIN {X -0.050,Y -607.463,Z 673.293,A 0.000,B 0.000,C 90.000,E1 88.740} C_DIS
LIN {X -0.226,Y -607.951,Z 673.284,A 0.000,B 0.000,C 90.000,E1 87.192} C_DIS
LIN {X -0.017,Y -608.088,Z 673.277,A 0.000,B 0.000,C 90.000,E1 85.869} C_DIS
LIN {X 0.144,Y -607.955,Z 673.270,A 0.000,B 0.000,C 90.000,E1 84.552} C_DIS
LIN {X 0.090,Y -607.714,Z 673.264,A 0.000,B 0.000,C 90.000,E1 83.514} C_DIS
LIN {X -0.247,Y -607.186,Z 673.257,A 0.000,B 0.000,C 90.000,E1 82.243} C_DIS
LIN {X -0.226,Y -606.636,Z 673.251,A 0.000,B 0.000,C 90.000,E1 81.197} C_DIS
LIN {X 0.062,Y -605.947,Z 673.247,A 0.000,B 0.000,C 90.000,E1 80.387} C_DIS
LIN {X 0.117,Y -604.388,Z 673.238,A 0.000,B 0.000,C 90.000,E1 78.814} C_DIS
LIN {X -0.056,Y -602.884,Z 673.231,A 0.000,B 0.000,C 90.000,E1 77.521} C_DIS
LIN {X 0.025,Y -601.533,Z 673.225,A 0.000,B 0.000,C 90.000,E1 76.464} C_DIS
LIN {X 0.079,Y -600.136,Z 673.219,A 0.000,B 0.000,C 90.000,E1 75.408} C_DIS
LIN {X 0.261,Y -598.589,Z 673.213,A 0.000,B 0.000,C 90.000,E1 74.338} C_DIS
LIN {X 0.126,Y -596.545,Z 673.206,A 0.000,B 0.000,C 90.000,E1 73.032} C_DIS
LIN {X -0.138,Y -594.743,Z 673.200,A 0.000,B 0.000,C 90.000,E1 72.000} C_DIS
LIN {X -0.167,Y -592.385,Z 673.193,A 0.000,B 0.000,C 90.000,E1 70.678} C_DIS
LIN {X -0.048,Y -589.711,Z 673.185,A 0.000,B 0.000,C 90.000,E1 69.337} C_DIS
LIN {X -0.190,Y -587.287,Z 673.179,A 0.000,B 0.000,C 90.000,E1 68.284} C_DIS
LIN {X -0.233,Y -585.263,Z 673.175,A 0.000,B 0.000,C 90.000,E1 67.486} C_DIS
LIN {X 0.333,Y -582.240,Z 673.169,A 0.000,B 0.000,C 90.000,E1 66.357} C_DIS
LIN {X 0.084,Y -578.875,Z 673.163,A 0.000,B 0.000,C 90.000,E1 65.305} C_DIS
LIN {X -0.345,Y -576.164,Z 673.158,A 0.000,B 0.000,C 90.000,E1 64.537} C_DIS
LIN {X -0.181,Y -572.181,Z 673.152,A 0.000,B 0.000,C 90.000,E1 63.435} C_DIS
LIN {X 0.007,Y -570.139,Z 673.149,A 0.000,B 0.000,C 90.000,E1 62.871} C_DIS
LIN {X 0.175,Y -566.210,Z 673.144,A 0.000,B 0.000,C 90.000,E1 61.897} C_DIS
LIN {X -0.283,Y -563.200,Z 673.140,A 0.000,B 0.000,C 90.000,E1 61.257} C_DIS
LIN {X -0.008,Y -559.898,Z 673.136,A 0.000,B 0.000,C 90.000,E1 60.539} C_DIS
LIN {X -0.251,Y -556.120,Z 673.133,A 0.000,B 0.000,C 90.000,E1 59.871} C_DIS
LIN {X -0.048,Y -551.810,Z 673.129,A 0.000,B 0.000,C 90.000,E1 59.154} C_DIS
LIN {X 0.012,Y -548.280,Z 673.126,A 0.000,B 0.000,C 90.000,E1 58.614} C_DIS
LIN {X -0.198,Y -544.266,Z 673.123,A 0.000,B 0.000,C 90.000,E1 58.074} C_DIS
LIN {X -0.145,Y -539.793,Z 673.119,A 0.000,B 0.000,C 90.000,E1 57.502} C_DIS
LIN {X 0.041,Y -534.875,Z 673.116,A 0.000,B 0.000,C 90.000,E1 56.914} C_DIS
LIN {X -0.017,Y -529.353,Z 673.113,A 0.000,B 0.000,C 90.000,E1 56.373} C_DIS
LIN {X -0.191,Y -524.948,Z 673.111,A 0.000,B 0.000,C 90.000,E1 56.008} C_DIS
LIN {X -0.073,Y -518.732,Z 673.108,A 0.000,B 0.000,C 90.000,E1 55.515} C_DIS
LIN {X 0.032,Y -512.339,Z 673.106,A 0.000,B 0.000,C 90.000,E1 55.055} C_DIS
LIN {X 0.007,Y -505.662,Z 673.104,A 0.000,B 0.000,C 90.000,E1 54.642} C_DIS
LIN {X 0.067,Y -497.357,Z 673.101,A 0.000,B 0.000,C 90.000,E1 54.149} C_DIS
LIN {X -0.019,Y -480.898,Z 673.096,A 0.000,B 0.000,C 90.000,E1 53.256} C_DIS
LIN {X 0.012,Y -466.131,Z 673.091,A 0.000,B 0.000,C 90.000,E1 52.431} C_DIS
LIN {X 0.098,Y -443.051,Z 673.084,A 0.000,B 0.000,C 90.000,E1 51.090} C_DIS
LIN {X 0.003,Y -434.940,Z 673.081,A 0.000,B 0.000,C 90.000,E1 50.598} C_DIS
LIN {X 0.124,Y -430.224,Z 673.079,A 0.000,B 0.000,C 90.000,E1 50.275} C_DIS
LIN {X 0.099,Y -430.174,Z 673.079,A 0.000,B 0.000,C 90.000,E1 50.275} C_DIS
LIN {X 0.082,Y -420.870,Z 673.056,A 0.000,B 0.000,C 90.000,E1 46.053} C_DIS
LIN {X -0.054,Y -418.378,Z 673.048,A 0.000,B 0.000,C 90.000,E1 44.717} C_DIS
LIN {X -0.107,Y -416.002,Z 673.043,A 0.000,B 0.000,C 90.000,E1 43.704} C_DIS
LIN {X -0.070,Y -416.019,Z 673.035,A 0.000,B 0.000,C 90.000,E1 42.243} C_DIS
LIN {X -0.041,Y -416.283,Z 673.021,A 0.000,B 0.000,C 90.000,E1 39.850} C_DIS
LIN {X 0.016,Y -417.580,Z 673.001,A 0.000,B 0.000,C 90.000,E1 36.091} C_DIS
LIN {X -0.056,Y -418.294,Z 672.993,A 0.000,B 0.000,C 90.000,E1 34.739} C_DIS
LIN {X 0.089,Y -419.508,Z 672.980,A 0.000,B 0.000,C 90.000,E1 32.339} C_DIS
LIN {X -0.104,Y -420.471,Z 672.970,A 0.000,B 0.000,C 90.000,E1 30.669} C_DIS
LIN {X 0.017,Y -421.769,Z 672.957,A 0.000,B 0.000,C 90.000,E1 28.281} C_DIS
LIN {X -0.047,Y -423.276,Z 672.944,A 0.000,B 0.000,C 90.000,E1 25.924} C_DIS
LIN {X 0.038,Y -426.988,Z 672.920,A 0.000,B 0.000,C 90.000,E1 21.535} C_DIS
LIN {X -0.011,Y -428.535,Z 672.910,A 0.000,B 0.000,C 90.000,E1 19.866} C_DIS
